REGION Network 17: ACTIVACION VAPOR VIVO Y SERPENTINA
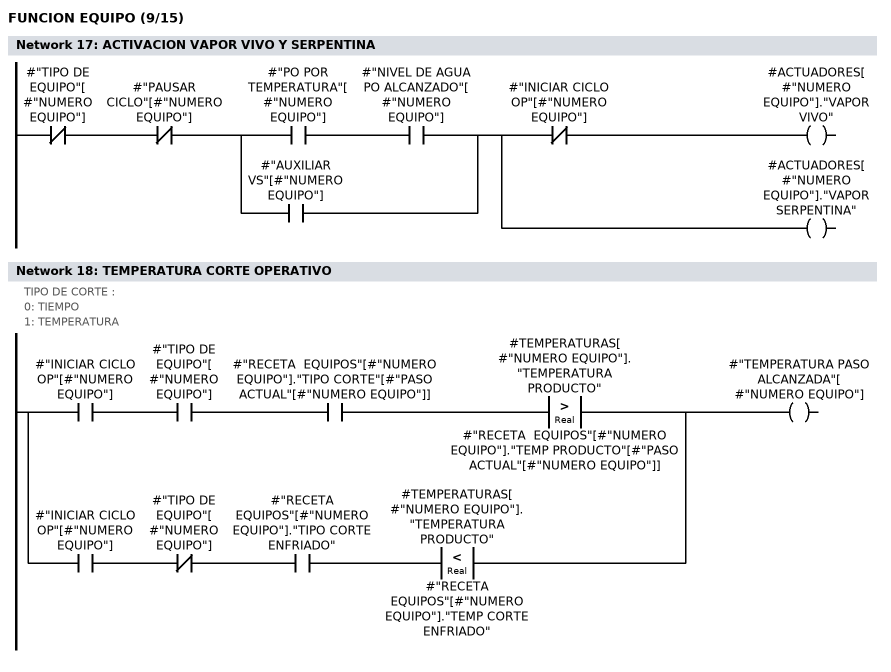
   RUNG wire#powerrail
      I_Contact( #"TIPO DE EQUIPO"[#"NUMERO EQUIPO"] )
      I_Contact( #"PAUSAR CICLO"[#"NUMERO EQUIPO"] )
      wire#w1
      Contact( #"PO POR TEMPERATURA"[#"NUMERO EQUIPO"] )
      Contact( #"NIVEL DE AGUA PO ALCANZADO"[#"NUMERO EQUIPO"] )
      wire#w2
      I_Contact( #"INICIAR CICLO OP"[#"NUMERO EQUIPO"] )
      Coil( #ACTUADORES[#"NUMERO EQUIPO"]."VAPOR VIVO" )
   END_RUNG
   RUNG wire#w1
      Contact( #"AUXILIAR VS"[#"NUMERO EQUIPO"] )
   END_RUNG wire#w2
   RUNG wire#w2
      Coil( #ACTUADORES[#"NUMERO EQUIPO"]."VAPOR SERPENTINA" )
   END_RUNG
   // the same network as SCL:
   #_w1 := NOT #"TIPO DE EQUIPO"[#"NUMERO EQUIPO"] AND NOT #"PAUSAR CICLO"[#"NUMERO EQUIPO"] AND ((#"PO POR TEMPERATURA"[#"NUMERO EQUIPO"] AND #"NIVEL DE AGUA PO ALCANZADO"[#"NUMERO EQUIPO"]) OR #"AUXILIAR VS"[#"NUMERO EQUIPO"]);
   #ACTUADORES[#"NUMERO EQUIPO"]."VAPOR VIVO" := #_w1 AND NOT #"INICIAR CICLO OP"[#"NUMERO EQUIPO"];
   #ACTUADORES[#"NUMERO EQUIPO"]."VAPOR SERPENTINA" := #_w1;
END_REGION

REGION Network 18: TEMPERATURA CORTE OPERATIVO
   // TIPO DE CORTE :
   // 
   // 0: TIEMPO
   // 1: TEMPERATURA
   RUNG wire#powerrail
      Contact( #"INICIAR CICLO OP"[#"NUMERO EQUIPO"] )
      Contact( #"TIPO DE EQUIPO"[#"NUMERO EQUIPO"] )
      Contact( #"RECETA  EQUIPOS"[#"NUMERO EQUIPO"]."TIPO CORTE"[#"PASO ACTUAL"[#"NUMERO EQUIPO"]] )
      { S7_Templates := "SrcType := Real" } GT_Contact(in1 := #TEMPERATURAS[#"NUMERO EQUIPO"]."TEMPERATURA PRODUCTO", in2 := #"RECETA  EQUIPOS"[#"NUMERO EQUIPO"]."TEMP PRODUCTO"[#"PASO ACTUAL"[#"NUMERO EQUIPO"]])
      wire#w1
      Coil( #"TEMPERATURA PASO ALCANZADA"[#"NUMERO EQUIPO"] )
   END_RUNG
   RUNG wire#powerrail
      Contact( #"INICIAR CICLO OP"[#"NUMERO EQUIPO"] )
      I_Contact( #"TIPO DE EQUIPO"[#"NUMERO EQUIPO"] )
      Contact( #"RECETA  EQUIPOS"[#"NUMERO EQUIPO"]."TIPO CORTE ENFRIADO" )
      { S7_Templates := "SrcType := Real" } LT_Contact(in1 := #TEMPERATURAS[#"NUMERO EQUIPO"]."TEMPERATURA PRODUCTO", in2 := #"RECETA  EQUIPOS"[#"NUMERO EQUIPO"]."TEMP CORTE ENFRIADO")
   END_RUNG wire#w1
   // the same network as SCL:
   #"TEMPERATURA PASO ALCANZADA"[#"NUMERO EQUIPO"] := (#"INICIAR CICLO OP"[#"NUMERO EQUIPO"] AND #"TIPO DE EQUIPO"[#"NUMERO EQUIPO"] AND #"RECETA  EQUIPOS"[#"NUMERO EQUIPO"]."TIPO CORTE"[#"PASO ACTUAL"[#"NUMERO EQUIPO"]] AND (#TEMPERATURAS[#"NUMERO EQUIPO"]."TEMPERATURA PRODUCTO" > #"RECETA  EQUIPOS"[#"NUMERO EQUIPO"]."TEMP PRODUCTO"[#"PASO ACTUAL"[#"NUMERO EQUIPO"]])) OR (#"INICIAR CICLO OP"[#"NUMERO EQUIPO"] AND NOT #"TIPO DE EQUIPO"[#"NUMERO EQUIPO"] AND #"RECETA  EQUIPOS"[#"NUMERO EQUIPO"]."TIPO CORTE ENFRIADO" AND (#TEMPERATURAS[#"NUMERO EQUIPO"]."TEMPERATURA PRODUCTO" < #"RECETA  EQUIPOS"[#"NUMERO EQUIPO"]."TEMP CORTE ENFRIADO"));
END_REGION

REGION Network 19: TIEMPO DE CORTE OPERATIVO
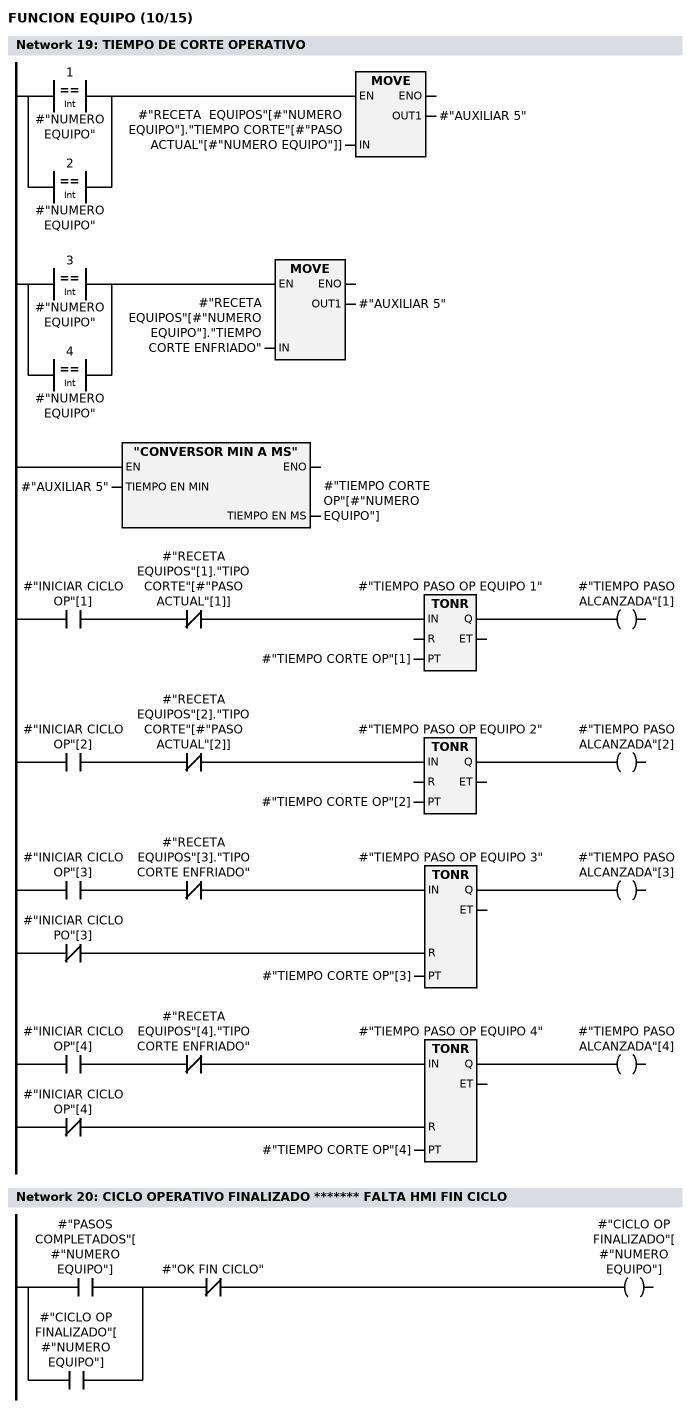
   IF (1 = #"NUMERO EQUIPO") OR (2 = #"NUMERO EQUIPO") THEN
       #"AUXILIAR 5" := #"RECETA  EQUIPOS"[#"NUMERO EQUIPO"]."TIEMPO CORTE"[#"PASO ACTUAL"[#"NUMERO EQUIPO"]];
   END_IF;
   IF (3 = #"NUMERO EQUIPO") OR (4 = #"NUMERO EQUIPO") THEN
       #"AUXILIAR 5" := #"RECETA  EQUIPOS"[#"NUMERO EQUIPO"]."TIEMPO CORTE ENFRIADO";
   END_IF;
   "CONVERSOR MIN A MS"("TIEMPO EN MIN" := #"AUXILIAR 5",
                        "TIEMPO EN MS" => #"TIEMPO CORTE OP"[#"NUMERO EQUIPO"]);
   #"TIEMPO PASO OP EQUIPO 1"(IN := #"INICIAR CICLO OP"[1] AND NOT #"RECETA  EQUIPOS"[1]."TIPO CORTE"[#"PASO ACTUAL"[1]],   // TONR
                           PT := #"TIEMPO CORTE OP"[1]);
   #"TIEMPO PASO ALCANZADA"[1] := #"TIEMPO PASO OP EQUIPO 1".Q;
   #"TIEMPO PASO OP EQUIPO 2"(IN := #"INICIAR CICLO OP"[2] AND NOT #"RECETA  EQUIPOS"[2]."TIPO CORTE"[#"PASO ACTUAL"[2]],   // TONR
                           PT := #"TIEMPO CORTE OP"[2]);
   #"TIEMPO PASO ALCANZADA"[2] := #"TIEMPO PASO OP EQUIPO 2".Q;
   #"TIEMPO PASO OP EQUIPO 3"(IN := #"INICIAR CICLO OP"[3] AND NOT #"RECETA  EQUIPOS"[3]."TIPO CORTE ENFRIADO",   // TONR
                           R := NOT #"INICIAR CICLO PO"[3],
                           PT := #"TIEMPO CORTE OP"[3]);
   #"TIEMPO PASO ALCANZADA"[3] := #"TIEMPO PASO OP EQUIPO 3".Q;
   #"TIEMPO PASO OP EQUIPO 4"(IN := #"INICIAR CICLO OP"[4] AND NOT #"RECETA  EQUIPOS"[4]."TIPO CORTE ENFRIADO",   // TONR
                           R := NOT #"INICIAR CICLO OP"[4],
                           PT := #"TIEMPO CORTE OP"[4]);
   #"TIEMPO PASO ALCANZADA"[4] := #"TIEMPO PASO OP EQUIPO 4".Q;
END_REGION

REGION Network 20: CICLO OPERATIVO FINALIZADO ******* FALTA HMI FIN CICLO
   RUNG wire#powerrail
      Contact( #"PASOS COMPLETADOS"[#"NUMERO EQUIPO"] )
      wire#w1
      I_Contact( #"OK FIN CICLO" )
      Coil( #"CICLO OP FINALIZADO"[#"NUMERO EQUIPO"] )
   END_RUNG
   RUNG wire#powerrail
      Contact( #"CICLO OP FINALIZADO"[#"NUMERO EQUIPO"] )
   END_RUNG wire#w1
   // the same network as SCL:
   #"CICLO OP FINALIZADO"[#"NUMERO EQUIPO"] := (#"PASOS COMPLETADOS"[#"NUMERO EQUIPO"] OR #"CICLO OP FINALIZADO"[#"NUMERO EQUIPO"]) AND NOT #"OK FIN CICLO";
END_REGION

REGION Network 21: CALCULO DE HISTERESIS
   // NIVEL OK
   // NIVEL BAJO
   // NIVEL ALTO
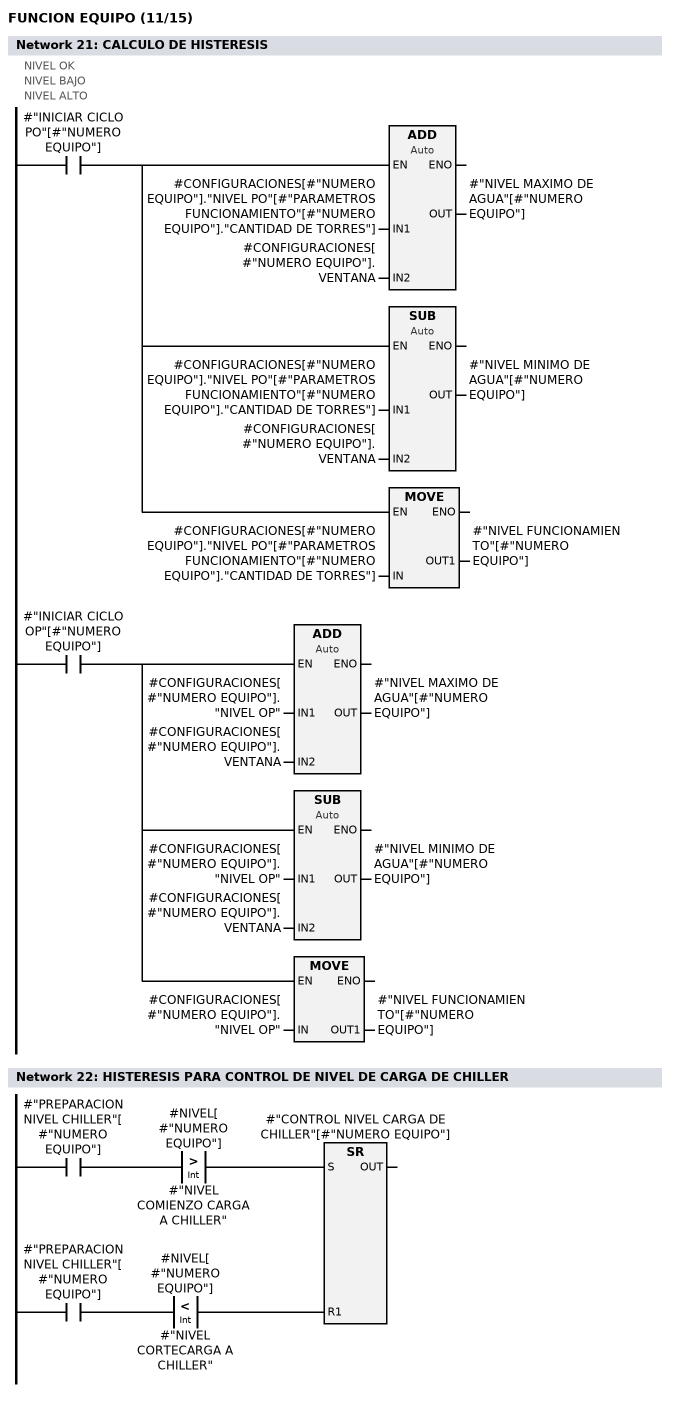
   RUNG wire#powerrail
      Contact( #"INICIAR CICLO PO"[#"NUMERO EQUIPO"] )
      wire#w1
      Add(in1 := #CONFIGURACIONES[#"NUMERO EQUIPO"]."NIVEL PO"[#"PARAMETROS FUNCIONAMIENTO"[#"NUMERO EQUIPO"]."CANTIDAD DE TORRES"], in2 := #CONFIGURACIONES[#"NUMERO EQUIPO"].VENTANA, out => #"NIVEL MAXIMO DE AGUA"[#"NUMERO EQUIPO"])
   END_RUNG
   RUNG wire#w1
      Sub(in1 := #CONFIGURACIONES[#"NUMERO EQUIPO"]."NIVEL PO"[#"PARAMETROS FUNCIONAMIENTO"[#"NUMERO EQUIPO"]."CANTIDAD DE TORRES"], in2 := #CONFIGURACIONES[#"NUMERO EQUIPO"].VENTANA, out => #"NIVEL MINIMO DE AGUA"[#"NUMERO EQUIPO"])
   END_RUNG
   RUNG wire#w1
      Move(in := #CONFIGURACIONES[#"NUMERO EQUIPO"]."NIVEL PO"[#"PARAMETROS FUNCIONAMIENTO"[#"NUMERO EQUIPO"]."CANTIDAD DE TORRES"], out1 => #"NIVEL FUNCIONAMIENTO"[#"NUMERO EQUIPO"])
   END_RUNG
   RUNG wire#powerrail
      Contact( #"INICIAR CICLO OP"[#"NUMERO EQUIPO"] )
      wire#w2
      Add(in1 := #CONFIGURACIONES[#"NUMERO EQUIPO"]."NIVEL OP", in2 := #CONFIGURACIONES[#"NUMERO EQUIPO"].VENTANA, out => #"NIVEL MAXIMO DE AGUA"[#"NUMERO EQUIPO"])
   END_RUNG
   RUNG wire#w2
      Sub(in1 := #CONFIGURACIONES[#"NUMERO EQUIPO"]."NIVEL OP", in2 := #CONFIGURACIONES[#"NUMERO EQUIPO"].VENTANA, out => #"NIVEL MINIMO DE AGUA"[#"NUMERO EQUIPO"])
   END_RUNG
   RUNG wire#w2
      Move(in := #CONFIGURACIONES[#"NUMERO EQUIPO"]."NIVEL OP", out1 => #"NIVEL FUNCIONAMIENTO"[#"NUMERO EQUIPO"])
   END_RUNG
   // the same network as SCL:
   #_w1 := #"INICIAR CICLO PO"[#"NUMERO EQUIPO"];
   IF #_w1 THEN
       #"NIVEL MAXIMO DE AGUA"[#"NUMERO EQUIPO"] := #CONFIGURACIONES[#"NUMERO EQUIPO"]."NIVEL PO"[#"PARAMETROS FUNCIONAMIENTO"[#"NUMERO EQUIPO"]."CANTIDAD DE TORRES"] + #CONFIGURACIONES[#"NUMERO EQUIPO"].VENTANA;
       #"NIVEL MINIMO DE AGUA"[#"NUMERO EQUIPO"] := #CONFIGURACIONES[#"NUMERO EQUIPO"]."NIVEL PO"[#"PARAMETROS FUNCIONAMIENTO"[#"NUMERO EQUIPO"]."CANTIDAD DE TORRES"] - #CONFIGURACIONES[#"NUMERO EQUIPO"].VENTANA;
       #"NIVEL FUNCIONAMIENTO"[#"NUMERO EQUIPO"] := #CONFIGURACIONES[#"NUMERO EQUIPO"]."NIVEL PO"[#"PARAMETROS FUNCIONAMIENTO"[#"NUMERO EQUIPO"]."CANTIDAD DE TORRES"];
   END_IF;
   #_w2 := #"INICIAR CICLO OP"[#"NUMERO EQUIPO"];
   IF #_w2 THEN
       #"NIVEL MAXIMO DE AGUA"[#"NUMERO EQUIPO"] := #CONFIGURACIONES[#"NUMERO EQUIPO"]."NIVEL OP" + #CONFIGURACIONES[#"NUMERO EQUIPO"].VENTANA;
       #"NIVEL MINIMO DE AGUA"[#"NUMERO EQUIPO"] := #CONFIGURACIONES[#"NUMERO EQUIPO"]."NIVEL OP" - #CONFIGURACIONES[#"NUMERO EQUIPO"].VENTANA;
       #"NIVEL FUNCIONAMIENTO"[#"NUMERO EQUIPO"] := #CONFIGURACIONES[#"NUMERO EQUIPO"]."NIVEL OP";
   END_IF;
END_REGION

REGION Network 22: HISTERESIS PARA CONTROL DE NIVEL DE CARGA DE CHILLER
   RUNG wire#powerrail
      Contact( #"PREPARACION NIVEL CHILLER"[#"NUMERO EQUIPO"] )
      { S7_Templates := "SrcType := Int" } GT_Contact(in1 := #NIVEL[#"NUMERO EQUIPO"], in2 := #"NIVEL COMIENZO CARGA A CHILLER")
      S_SR(operand := #"CONTROL NIVEL CARGA DE CHILLER"[#"NUMERO EQUIPO"], r1 := wire#w1)
   END_RUNG
   RUNG wire#powerrail
      Contact( #"PREPARACION NIVEL CHILLER"[#"NUMERO EQUIPO"] )
      { S7_Templates := "SrcType := Int" } LT_Contact(in1 := #NIVEL[#"NUMERO EQUIPO"], in2 := #"NIVEL CORTECARGA A CHILLER")
   END_RUNG wire#w1
   // the same network as SCL:
   #_w1 := #"PREPARACION NIVEL CHILLER"[#"NUMERO EQUIPO"] AND (#NIVEL[#"NUMERO EQUIPO"] < #"NIVEL CORTECARGA A CHILLER");
   IF #"PREPARACION NIVEL CHILLER"[#"NUMERO EQUIPO"] AND (#NIVEL[#"NUMERO EQUIPO"] > #"NIVEL COMIENZO CARGA A CHILLER") THEN
       #"CONTROL NIVEL CARGA DE CHILLER"[#"NUMERO EQUIPO"] := TRUE;   // SR flip-flop
   END_IF;
   IF #_w1 THEN #"CONTROL NIVEL CARGA DE CHILLER"[#"NUMERO EQUIPO"] := FALSE; END_IF;
END_REGION

REGION Network 23: CONTROL DE NIVEL DE AGUA DE TANQUE
   // LO CONTROLO CON UN SET Y RESET
   // 
   // 1 SR : BOMBA EGRESO
   // 2 SR : BOMBA INGRESO
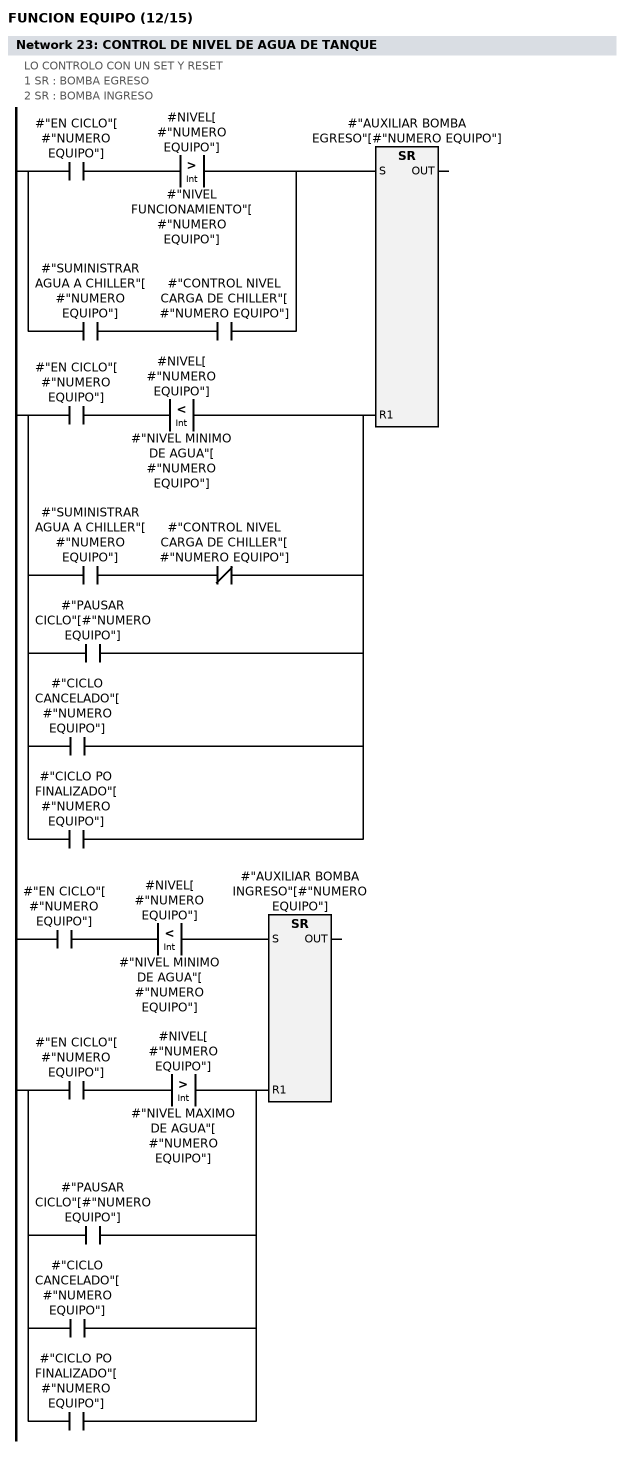
   RUNG wire#powerrail
      Contact( #"EN CICLO"[#"NUMERO EQUIPO"] )
      { S7_Templates := "SrcType := Int" } GT_Contact(in1 := #NIVEL[#"NUMERO EQUIPO"], in2 := #"NIVEL FUNCIONAMIENTO"[#"NUMERO EQUIPO"])
      wire#w1
      S_SR(operand := #"AUXILIAR BOMBA EGRESO"[#"NUMERO EQUIPO"], r1 := wire#w2)
   END_RUNG
   RUNG wire#powerrail
      Contact( #"SUMINISTRAR AGUA A CHILLER"[#"NUMERO EQUIPO"] )
      Contact( #"CONTROL NIVEL CARGA DE CHILLER"[#"NUMERO EQUIPO"] )
   END_RUNG wire#w1
   RUNG wire#powerrail
      Contact( #"EN CICLO"[#"NUMERO EQUIPO"] )
      { S7_Templates := "SrcType := Int" } LT_Contact(in1 := #NIVEL[#"NUMERO EQUIPO"], in2 := #"NIVEL MINIMO DE AGUA"[#"NUMERO EQUIPO"])
   END_RUNG wire#w2
   RUNG wire#powerrail
      Contact( #"SUMINISTRAR AGUA A CHILLER"[#"NUMERO EQUIPO"] )
      I_Contact( #"CONTROL NIVEL CARGA DE CHILLER"[#"NUMERO EQUIPO"] )
   END_RUNG wire#w2
   RUNG wire#powerrail
      Contact( #"PAUSAR CICLO"[#"NUMERO EQUIPO"] )
   END_RUNG wire#w2
   RUNG wire#powerrail
      Contact( #"CICLO CANCELADO"[#"NUMERO EQUIPO"] )
   END_RUNG wire#w2
   RUNG wire#powerrail
      Contact( #"CICLO PO FINALIZADO"[#"NUMERO EQUIPO"] )
   END_RUNG wire#w2
   RUNG wire#powerrail
      Contact( #"EN CICLO"[#"NUMERO EQUIPO"] )
      { S7_Templates := "SrcType := Int" } LT_Contact(in1 := #NIVEL[#"NUMERO EQUIPO"], in2 := #"NIVEL MINIMO DE AGUA"[#"NUMERO EQUIPO"])
      S_SR(operand := #"AUXILIAR BOMBA INGRESO"[#"NUMERO EQUIPO"], r1 := wire#w3)
   END_RUNG
   RUNG wire#powerrail
      Contact( #"EN CICLO"[#"NUMERO EQUIPO"] )
      { S7_Templates := "SrcType := Int" } GT_Contact(in1 := #NIVEL[#"NUMERO EQUIPO"], in2 := #"NIVEL MAXIMO DE AGUA"[#"NUMERO EQUIPO"])
   END_RUNG wire#w3
   RUNG wire#powerrail
      Contact( #"PAUSAR CICLO"[#"NUMERO EQUIPO"] )
   END_RUNG wire#w3
   RUNG wire#powerrail
      Contact( #"CICLO CANCELADO"[#"NUMERO EQUIPO"] )
   END_RUNG wire#w3
   RUNG wire#powerrail
      Contact( #"CICLO PO FINALIZADO"[#"NUMERO EQUIPO"] )
   END_RUNG wire#w3
   // the same network as SCL:
   #_w1 := (#"EN CICLO"[#"NUMERO EQUIPO"] AND (#NIVEL[#"NUMERO EQUIPO"] < #"NIVEL MINIMO DE AGUA"[#"NUMERO EQUIPO"])) OR (#"SUMINISTRAR AGUA A CHILLER"[#"NUMERO EQUIPO"] AND NOT #"CONTROL NIVEL CARGA DE CHILLER"[#"NUMERO EQUIPO"]) OR #"PAUSAR CICLO"[#"NUMERO EQUIPO"] OR #"CICLO CANCELADO"[#"NUMERO EQUIPO"] OR #"CICLO PO FINALIZADO"[#"NUMERO EQUIPO"];
   IF (#"EN CICLO"[#"NUMERO EQUIPO"] AND (#NIVEL[#"NUMERO EQUIPO"] > #"NIVEL FUNCIONAMIENTO"[#"NUMERO EQUIPO"])) OR (#"SUMINISTRAR AGUA A CHILLER"[#"NUMERO EQUIPO"] AND #"CONTROL NIVEL CARGA DE CHILLER"[#"NUMERO EQUIPO"]) THEN
       #"AUXILIAR BOMBA EGRESO"[#"NUMERO EQUIPO"] := TRUE;   // SR flip-flop
   END_IF;
   IF #_w1 THEN #"AUXILIAR BOMBA EGRESO"[#"NUMERO EQUIPO"] := FALSE; END_IF;
   #_w2 := (#"EN CICLO"[#"NUMERO EQUIPO"] AND (#NIVEL[#"NUMERO EQUIPO"] > #"NIVEL MAXIMO DE AGUA"[#"NUMERO EQUIPO"])) OR #"PAUSAR CICLO"[#"NUMERO EQUIPO"] OR #"CICLO CANCELADO"[#"NUMERO EQUIPO"] OR #"CICLO PO FINALIZADO"[#"NUMERO EQUIPO"];
   IF #"EN CICLO"[#"NUMERO EQUIPO"] AND (#NIVEL[#"NUMERO EQUIPO"] < #"NIVEL MINIMO DE AGUA"[#"NUMERO EQUIPO"]) THEN
       #"AUXILIAR BOMBA INGRESO"[#"NUMERO EQUIPO"] := TRUE;   // SR flip-flop
   END_IF;
   IF #_w2 THEN #"AUXILIAR BOMBA INGRESO"[#"NUMERO EQUIPO"] := FALSE; END_IF;
END_REGION

REGION Network 24: DELAY ENTRE VALVULAS Y BOMBAS DE INGRESO Y EGRESO
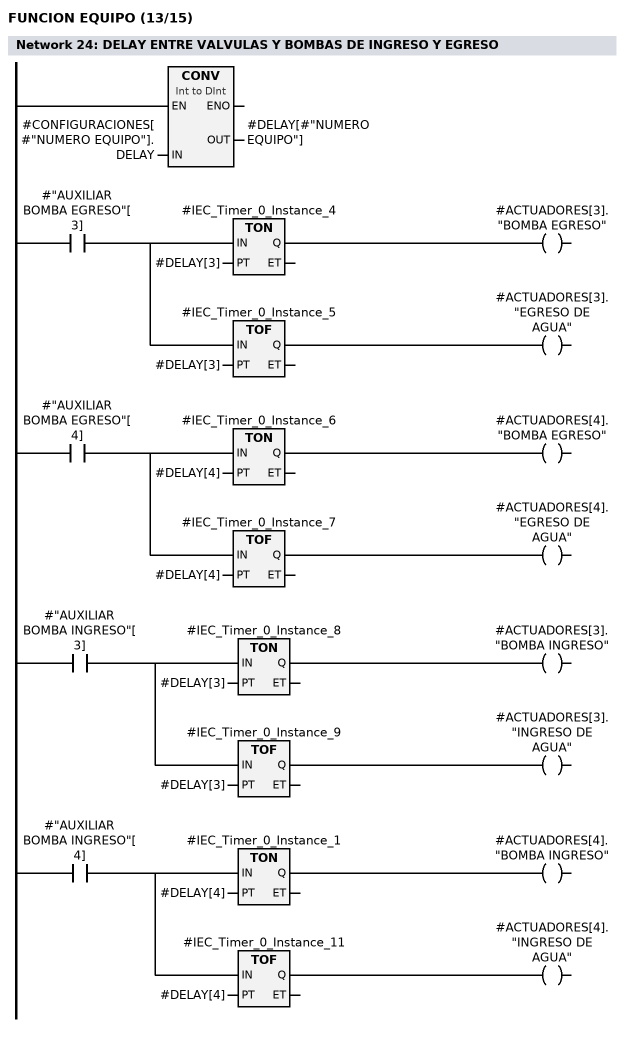
   #DELAY[#"NUMERO EQUIPO"] := INT_TO_DINT(#CONFIGURACIONES[#"NUMERO EQUIPO"].DELAY);
   #IEC_Timer_0_Instance_4(IN := #"AUXILIAR BOMBA EGRESO"[3], PT := #DELAY[3]);   // TON
   #ACTUADORES[3]."BOMBA EGRESO" := #IEC_Timer_0_Instance_4.Q;
   #IEC_Timer_0_Instance_5(IN := #"AUXILIAR BOMBA EGRESO"[3], PT := #DELAY[3]);   // TOF
   #ACTUADORES[3]."EGRESO DE AGUA" := #IEC_Timer_0_Instance_5.Q;
   #IEC_Timer_0_Instance_6(IN := #"AUXILIAR BOMBA EGRESO"[4], PT := #DELAY[4]);   // TON
   #ACTUADORES[4]."BOMBA EGRESO" := #IEC_Timer_0_Instance_6.Q;
   #IEC_Timer_0_Instance_7(IN := #"AUXILIAR BOMBA EGRESO"[4], PT := #DELAY[4]);   // TOF
   #ACTUADORES[4]."EGRESO DE AGUA" := #IEC_Timer_0_Instance_7.Q;
   #IEC_Timer_0_Instance_8(IN := #"AUXILIAR BOMBA INGRESO"[3], PT := #DELAY[3]);   // TON
   #ACTUADORES[3]."BOMBA INGRESO" := #IEC_Timer_0_Instance_8.Q;
   #IEC_Timer_0_Instance_9(IN := #"AUXILIAR BOMBA INGRESO"[3], PT := #DELAY[3]);   // TOF
   #ACTUADORES[3]."INGRESO DE AGUA" := #IEC_Timer_0_Instance_9.Q;
   #IEC_Timer_0_Instance_1(IN := #"AUXILIAR BOMBA INGRESO"[4], PT := #DELAY[4]);   // TON
   #ACTUADORES[4]."BOMBA INGRESO" := #IEC_Timer_0_Instance_1.Q;
   #IEC_Timer_0_Instance_11(IN := #"AUXILIAR BOMBA INGRESO"[4], PT := #DELAY[4]);   // TOF
   #ACTUADORES[4]."INGRESO DE AGUA" := #IEC_Timer_0_Instance_11.Q;
END_REGION

REGION Network 25: NIVELES DE CHILLER
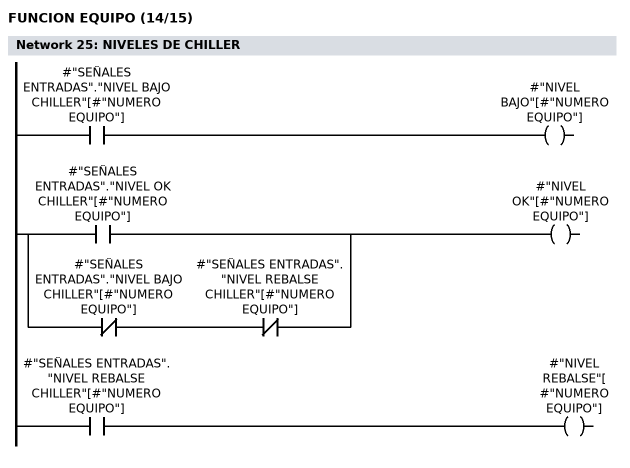
   RUNG wire#powerrail
      Contact( #"SEÑALES ENTRADAS"."NIVEL BAJO CHILLER"[#"NUMERO EQUIPO"] )
      Coil( #"NIVEL BAJO"[#"NUMERO EQUIPO"] )
   END_RUNG
   RUNG wire#powerrail
      Contact( #"SEÑALES ENTRADAS"."NIVEL OK CHILLER"[#"NUMERO EQUIPO"] )
      wire#w1
      Coil( #"NIVEL OK"[#"NUMERO EQUIPO"] )
   END_RUNG
   RUNG wire#powerrail
      I_Contact( #"SEÑALES ENTRADAS"."NIVEL BAJO CHILLER"[#"NUMERO EQUIPO"] )
      I_Contact( #"SEÑALES ENTRADAS"."NIVEL REBALSE CHILLER"[#"NUMERO EQUIPO"] )
   END_RUNG wire#w1
   RUNG wire#powerrail
      Contact( #"SEÑALES ENTRADAS"."NIVEL REBALSE CHILLER"[#"NUMERO EQUIPO"] )
      Coil( #"NIVEL REBALSE"[#"NUMERO EQUIPO"] )
   END_RUNG
   // the same network as SCL:
   #"NIVEL BAJO"[#"NUMERO EQUIPO"] := #"SEÑALES ENTRADAS"."NIVEL BAJO CHILLER"[#"NUMERO EQUIPO"];
   #"NIVEL OK"[#"NUMERO EQUIPO"] := #"SEÑALES ENTRADAS"."NIVEL OK CHILLER"[#"NUMERO EQUIPO"] OR (NOT #"SEÑALES ENTRADAS"."NIVEL BAJO CHILLER"[#"NUMERO EQUIPO"] AND NOT #"SEÑALES ENTRADAS"."NIVEL REBALSE CHILLER"[#"NUMERO EQUIPO"]);
   #"NIVEL REBALSE"[#"NUMERO EQUIPO"] := #"SEÑALES ENTRADAS"."NIVEL REBALSE CHILLER"[#"NUMERO EQUIPO"];
END_REGION

REGION Network 26: PASE DE ESTADOS
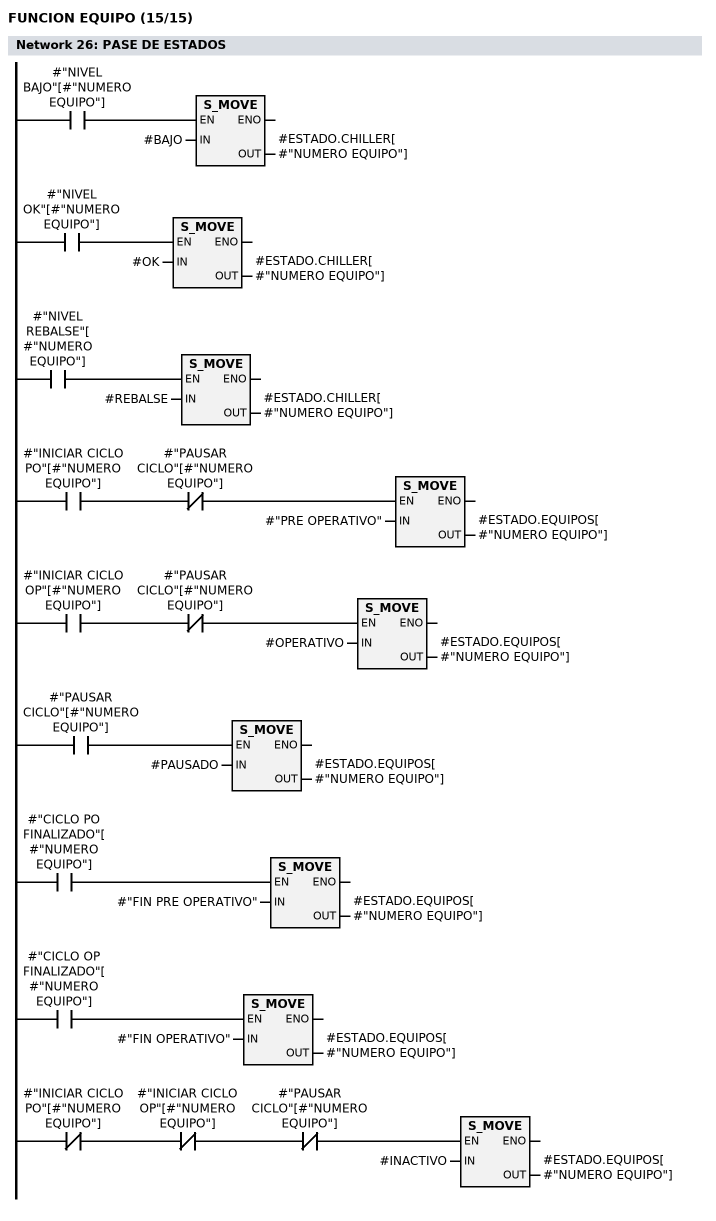
   RUNG wire#powerrail
      Contact( #"NIVEL BAJO"[#"NUMERO EQUIPO"] )
      S_Move(in := #BAJO, out => #ESTADO.CHILLER[#"NUMERO EQUIPO"])
   END_RUNG
   RUNG wire#powerrail
      Contact( #"NIVEL OK"[#"NUMERO EQUIPO"] )
      S_Move(in := #OK, out => #ESTADO.CHILLER[#"NUMERO EQUIPO"])
   END_RUNG
   RUNG wire#powerrail
      Contact( #"NIVEL REBALSE"[#"NUMERO EQUIPO"] )
      S_Move(in := #REBALSE, out => #ESTADO.CHILLER[#"NUMERO EQUIPO"])
   END_RUNG
   RUNG wire#powerrail
      Contact( #"INICIAR CICLO PO"[#"NUMERO EQUIPO"] )
      I_Contact( #"PAUSAR CICLO"[#"NUMERO EQUIPO"] )
      S_Move(in := #"PRE OPERATIVO", out => #ESTADO.EQUIPOS[#"NUMERO EQUIPO"])
   END_RUNG
   RUNG wire#powerrail
      Contact( #"INICIAR CICLO OP"[#"NUMERO EQUIPO"] )
      I_Contact( #"PAUSAR CICLO"[#"NUMERO EQUIPO"] )
      S_Move(in := #OPERATIVO, out => #ESTADO.EQUIPOS[#"NUMERO EQUIPO"])
   END_RUNG
   RUNG wire#powerrail
      Contact( #"PAUSAR CICLO"[#"NUMERO EQUIPO"] )
      S_Move(in := #PAUSADO, out => #ESTADO.EQUIPOS[#"NUMERO EQUIPO"])
   END_RUNG
   RUNG wire#powerrail
      Contact( #"CICLO PO FINALIZADO"[#"NUMERO EQUIPO"] )
      S_Move(in := #"FIN PRE OPERATIVO", out => #ESTADO.EQUIPOS[#"NUMERO EQUIPO"])
   END_RUNG
   RUNG wire#powerrail
      Contact( #"CICLO OP FINALIZADO"[#"NUMERO EQUIPO"] )
      S_Move(in := #"FIN OPERATIVO", out => #ESTADO.EQUIPOS[#"NUMERO EQUIPO"])
   END_RUNG
   RUNG wire#powerrail
      I_Contact( #"INICIAR CICLO PO"[#"NUMERO EQUIPO"] )
      I_Contact( #"INICIAR CICLO OP"[#"NUMERO EQUIPO"] )
      I_Contact( #"PAUSAR CICLO"[#"NUMERO EQUIPO"] )
      S_Move(in := #INACTIVO, out => #ESTADO.EQUIPOS[#"NUMERO EQUIPO"])
   END_RUNG
   // the same network as SCL:
   IF #"NIVEL BAJO"[#"NUMERO EQUIPO"] THEN #ESTADO.CHILLER[#"NUMERO EQUIPO"] := #BAJO; END_IF;
   IF #"NIVEL OK"[#"NUMERO EQUIPO"] THEN #ESTADO.CHILLER[#"NUMERO EQUIPO"] := #OK; END_IF;
   IF #"NIVEL REBALSE"[#"NUMERO EQUIPO"] THEN #ESTADO.CHILLER[#"NUMERO EQUIPO"] := #REBALSE; END_IF;
   IF #"INICIAR CICLO PO"[#"NUMERO EQUIPO"] AND NOT #"PAUSAR CICLO"[#"NUMERO EQUIPO"] THEN
       #ESTADO.EQUIPOS[#"NUMERO EQUIPO"] := #"PRE OPERATIVO";
   END_IF;
   IF #"INICIAR CICLO OP"[#"NUMERO EQUIPO"] AND NOT #"PAUSAR CICLO"[#"NUMERO EQUIPO"] THEN
       #ESTADO.EQUIPOS[#"NUMERO EQUIPO"] := #OPERATIVO;
   END_IF;
   IF #"PAUSAR CICLO"[#"NUMERO EQUIPO"] THEN #ESTADO.EQUIPOS[#"NUMERO EQUIPO"] := #PAUSADO; END_IF;
   IF #"CICLO PO FINALIZADO"[#"NUMERO EQUIPO"] THEN
       #ESTADO.EQUIPOS[#"NUMERO EQUIPO"] := #"FIN PRE OPERATIVO";
   END_IF;
   IF #"CICLO OP FINALIZADO"[#"NUMERO EQUIPO"] THEN
       #ESTADO.EQUIPOS[#"NUMERO EQUIPO"] := #"FIN OPERATIVO";
   END_IF;
   IF NOT #"INICIAR CICLO PO"[#"NUMERO EQUIPO"] AND NOT #"INICIAR CICLO OP"[#"NUMERO EQUIPO"] AND NOT #"PAUSAR CICLO"[#"NUMERO EQUIPO"] THEN
       #ESTADO.EQUIPOS[#"NUMERO EQUIPO"] := #INACTIVO;
   END_IF;
END_REGION
END_FUNCTION_BLOCK

FUNCTION_BLOCK "COCINA"   // FB5, LAD
{ S7_Optimized_Access := 'TRUE' }
VERSION : 0.1
   VAR_INPUT
      REARME : Bool;
      "PARAMETROS CICLOS" : Struct
         "CANTIDAD DE TORRES" : Int;
         "NIVEL MINIMO" : Array[1..3] of Int;   // El arreglo es porque hay 3 torres
         "TIPO DE CORTE" : Bool;
         "TEMPERATURA CORTE PO" : Int;
         "TIEMPO CORTE PO" : Int;
         "NUMERO RECETA" : Int;
         "NOMBRE RECETA" : String;
         "ESTADO ACTUAL" : String;
         "TIEMPO TOTAL TRANSCURRIDO" : Int;
         "PASO ACTUAL" : Int;
         "VAPOR VIVO" : Bool;
      END_STRUCT;
      CONFIGURACION : Struct
         DELAY : Int;
         HISTERESIS : DInt;
         "TIEMPO MAXIMO CICLO" : Int;
         "NIVEL CRITICO" : Int;
         "NIVEL PO" : Array[1..3] of Int;
         "NIVEL OP" : Int;
         VENTANA : Int;
         "NIVEL CRITICO OP" : Int;
      END_STRUCT;
      RECETA : Struct
         PASOS : Int;
         "TEMP AGUA" : Array[1..4] of Int;
         "TEMP PRODUCTO" : Array[1..4] of Int;
         "TIEMPO CORTE" : Array[1..4] of Int;
         "TIPO CORTE" : Array[1..4] of Bool;
         NOMBRE : String;
         "TIEMPO CORTE ENFRIADO" : Int;
         "TEMP CORTE ENFRIADO" : Int;
         "TIPO CORTE ENFRIADO" : Bool;
      END_STRUCT;
      TEMPERATURAS : Struct
         "TEMPERATURA AGUA" : Real;
         "TEMPERATURA INGRESO" : Real;
         "TEMPERATURA PRODUCTO" : Real;
         "TEMPERATURA AGUA SC" : Real;
         "TEMPERATURA INGRESO SC" : Real;
         "TEMPERATURA PRODUCTO SC" : Real;
      END_STRUCT;
      NIVEL : Int;
      GUARDAMOTOR : Bool;
      "VAPOR VIVO CERRADO" : Bool;
      "VAPOR VIVO ABIERTO" : Bool;
      "SERPENTINA CERRADA" : Bool;
      "SERPENTINA ABIERTA" : Bool;
      "MANUAL VAPOR VIVO" : Bool;
      "MANUAL VAPOR SERPENTINA" : Bool;
      "MANUAL CARGA DE AGUA" : Bool;
      "MANUAL TOMA FILTRO" : Bool;
      "MANUAL BOMBA" : Bool;
      "MANUAL BALIZA VERDE" : Bool;
      "MANUAL BALIZA ROJA" : Bool;
      "MANUAL LEVANTAR TAPA" : Bool;
      "MANUAL BAJAR TAPA" : Bool;
      "EQUIPO SELECCIONADO" : Int;
      "NUMERO DE EQUIPO" : Int;
      "SALTAR PASO" : Bool;
      "INICIAR PRE OPERATIVO" : Bool;
      "INICIAR OPERATIVO" : Bool;
      PAUSA : Bool;
      CONTINUAR : Bool;
      CANCELAR : Bool;
      "PULSADOR EMERGENCIA" : Bool;
      "OK FIN CICLO" : Bool;
      "OK CANCELAR" : Bool;
      "RESET ACTUADORES MANUAL" : Bool;
      "CONFIRMAR LOTE" : Bool;
   END_VAR
   VAR_OUTPUT
      "BALIZA VERDE" : Bool;
      "BALIZA ROJA" : Bool;
      BUZER : Bool;
      BOMBA : Bool;
      "CARGA DE AGUA" : Bool;
      "TOMA FILTRO" : Bool;
      "VAPOR SERPENTINA" : Bool;
      "VAPOR VIVO" : Bool;
      ESTADO : Struct
         EQUIPO : String;
         CHILLER : String;
         "COLOR EN HMI" : Int;
         "TIEMPO TRANSCURRIDO" : DInt;
         "EN PO" : Bool;
         "EN OP" : Bool;
         "EN CICLO" : Bool;
         "TIPO DE CORTE" : String;
         "PULSADOR PAUSA" : Bool;
         "PULSADOR CONTINUAR" : Bool;
         "PULSADOR CANCELAR" : Bool;
         "CICLO CANCELADO" : Bool;
         "CICLO FINALIZADO" : Bool;
         "PULSADOR CICLO CANCELADO" : Bool;
         "PULSADOR CICLO FINALIZADO" : Bool;
         "RESET ACTUADORES" : Bool;
         "MANUAL ACTIVO" : Bool;
         "PASO ACTUAL" : Int;
         "CONFIRMACION LOTE" : Bool;
      END_STRUCT;
      ALARMAS : Struct
         "FALLA VALVULA VAPOR SERPENTINA" : Bool;
         "FALLA VALVULA VAPOR VIVO" : Bool;
         "FALLA GUARDAMOTOR" : Bool;
         "NIVEL CRITICO" : Bool;
         "FALLA SENSOR TEMP AGUA" : Bool;
         "FALLA SENSOR TEMP INGRESO" : Bool;
         "FALLA SENSOR TEMP PRODUCTO" : Bool;
         "TIEMPO MAXIMO CARGA DE AGUA" : Bool;
      END_STRUCT;
      "ESTADO SALIDAS" : Struct
         "BALIZA VERDE" : Bool;
         "BALIZA ROJA" : Bool;
         BOMBA : Bool;
         "CARGA DE GUA" : Bool;
         "TOMA FILTRO" : Bool;
         "VAPOR SERPENTINA" : Bool;
         "VAPOR VIVO" : Bool;
      END_STRUCT;
      "ESTADO ENTRADAS" : Struct
         GUARDAMOTOR : Bool;
         "VAPOR VIVO CERRADO" : Bool;
         "VAPOR VIVO ABIERTO" : Bool;
         "SERPENTINA CERRADA" : Bool;
         "SERPENTINA ABIERTA" : Bool;
      END_STRUCT;
   END_VAR
   VAR
      HABILITADO : Bool;
      "EN FALLA" : Bool;
      "CICLO CANCELADO" : Bool;
      "CICLO PAUSADO" : Bool;
      "CICLO PO ACTIVO" : Bool;
      "CICLO OP ACTIVO" : Bool;
      "FIN CICLO PO" : Bool;
      "NIVEL PO" : Int;
      "NIVEL TQ ALCANZADO" : Bool;
      "CARGA AGUA TQ" : Bool;
      "NIVEL PARA CARGA DE AGUA" : Int;
      "TEMPERATURA PO ALCANZADA" : Bool;
      "TIEMPO PO ALCANZADO" : Bool;
      "TIEMPO CORTE PO" : DInt;
      IEC_Timer_0_Instance : TONR_TIME;
      "FIN CICLO OP" : Bool;
      IEC_Counter_0_Instance : CTU_INT;
      "PASO ACTUAL" : Int;
      AUXILIAR : Int;
      "TEMPERATURA PASO ALCANZADA" : Bool;
      IEC_Timer_0_Instance_1 : TONR_TIME;
      "TIEMPO PASO ALCANZADO" : Bool;
      "TIEMPO DE PASO EN OP" : DInt;
      "TEMP MAXIMA" : Real;
      "TEMP MINIMA" : Real;
      "TEMP EN RANGO" : Bool;
      "TEMP BAJA" : Bool;
      "TEMP ALTA" : Bool;
      "CICLO PO FINALIZADO" : Bool;
      "CICLO OP FINALIZADO" : Bool;
      IEC_Timer_0_Instance_2 : TON_TIME;
      IEC_Timer_0_Instance_3 : TON_TIME;
      "FALLA VALVULA SERPENTINA" : Bool;
      "FALLA CIERRE VS" : Bool;
      "FALLA VALVULA VAPOR VIVO" : Bool;
      "FALLA CIERRE VV" : Bool;
      IEC_Timer_0_Instance_4 : TON_TIME;
      IEC_Timer_0_Instance_5 : TON_TIME;
      "SE ALCANZO UN NIVEL CRITICO" : Bool;
      F1 : Bool;
      "FALLA SENSOR TEMPERATURA" : Bool;
      IEC_Timer_0_Instance_6 : TONR_TIME;
      IEC_Timer_0_Instance_7 : TON_TIME;
      IEC_Timer_0_Instance_8 : TON_TIME;
      IEC_Timer_0_Instance_9 : TONR_TIME;
      "TIEMPO MAXIMO" : DInt;
      "AUXILIAR TIEMPO" : DInt;
      IEC_Timer_0_Instance_10 : TONR_TIME;
      "TIEMPO MAXIMO CARGA DE AGUA" : Bool;
      "NIVEL CRITICO PO" : Bool;
      "NIVEL CRITICO OP" : Bool;
      "CONTINUAR CICLO" : Bool;
      IEC_Timer_0_Instance_11 : TOF_TIME;
      F5 : Bool;
      F6 : Bool;
      F7 : Bool;
      F8 : Bool;
      "TEMP MAXIMA CHILLER" : Real;
      "TEMP MINIMA CHILLER" : Real;
      "TEMP ALTA CHILLER" : Bool;
      "TEMP BAJA CHILLER" : Bool;
      "TEMP EN RANGO CHILLER" : Bool;
      IEC_Timer_0_Instance_12 : TOF_TIME;
      F9 : Bool;
      "PREPARACION FRIO CHILLER EN COCCION" : Bool;
      "PREPARACION FRIO CHILLER EN ENFRIADO" : Bool;
      "SALIDA AUX 1 CLIENTE" : Bool;
      "SALIDA AUX 2 CLIENTE" : Bool;
      "CONFIRMAR LOTE_1" : Bool;
   END_VAR
   VAR CONSTANT
      "MAXIMO APERTURA VALVULAS" : Time := T#7S;
      TEMPERATURA : String := 'TEMPERATURA';
      TIEMPO : String := 'TIEMPO';
      "PRE OPERACIONAL" : String := 'PRE OPERACIONAL';
      OPERACIONAL : String := 'OPERACIONAL';
      PAUSADO : String := 'PAUSADO';
      INACTIVO : String := 'INACTIVO';
      CANCELADO : String := 'CANCELADO';
      FINALIZADO : String := 'FINALIZADO';
      "NIVEL FILTRO" : Int := 980;
      "NIVEL TOMA FILTRO" : Int := 550;
   END_VAR
   VAR_TEMP   // added for the SCL form of the ladder/FBD networks
      _w1 : Bool;
      _w2 : Bool;
      _w3 : Bool;
      _w4 : Bool;
      _w5 : Bool;
   END_VAR
   // // CONFIGURACION."NIVEL PO"[1] : Nivel PO para 1 torre
   // // CONFIGURACION."NIVEL PO"[2] : Nivel PO para 2 torres
   // // CONFIGURACION."NIVEL PO"[3] : Nivel PO para 3 torres
BEGIN

REGION Network 1: HABILITACION
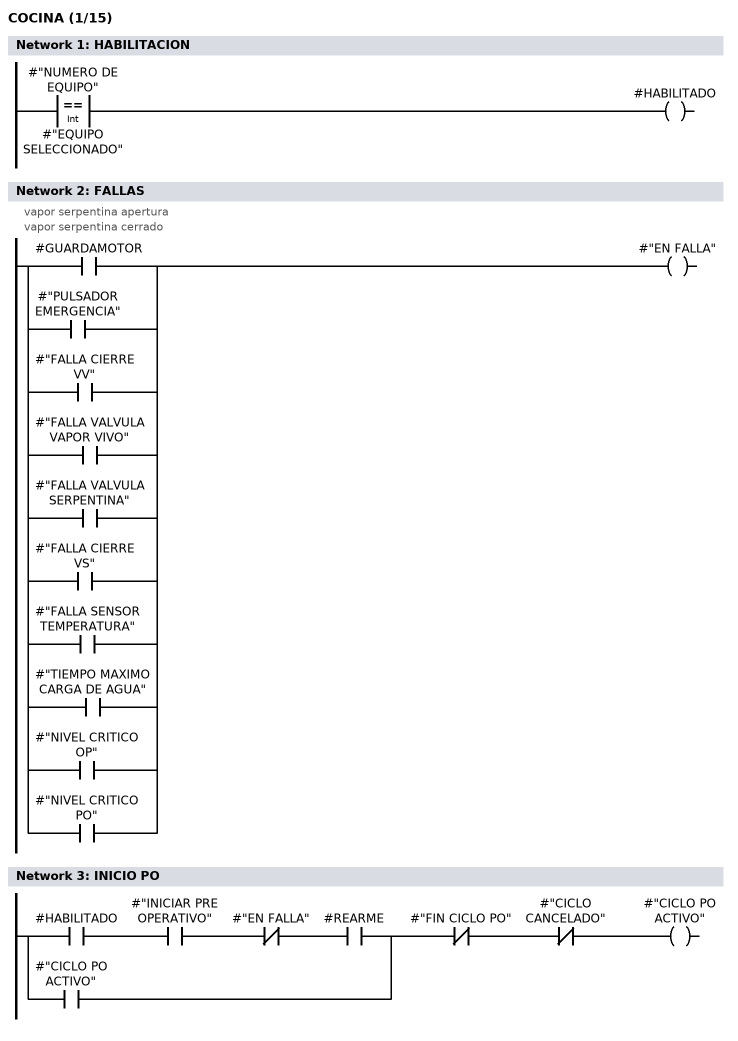
   RUNG wire#powerrail
      { S7_Templates := "SrcType := Int" } EQ_Contact(in1 := #"NUMERO DE EQUIPO", in2 := #"EQUIPO SELECCIONADO")
      Coil( #HABILITADO )
   END_RUNG
   // the same network as SCL:
   #HABILITADO := #"NUMERO DE EQUIPO" = #"EQUIPO SELECCIONADO";
END_REGION

REGION Network 2: FALLAS
   // vapor serpentina apertura
   // vapor serpentina cerrado
   RUNG wire#powerrail
      Contact( #GUARDAMOTOR )
      wire#w1
      Coil( #"EN FALLA" )
   END_RUNG
   RUNG wire#powerrail
      Contact( #"PULSADOR EMERGENCIA" )
   END_RUNG wire#w1
   RUNG wire#powerrail
      Contact( #"FALLA CIERRE VV" )
   END_RUNG wire#w1
   RUNG wire#powerrail
      Contact( #"FALLA VALVULA VAPOR VIVO" )
   END_RUNG wire#w1
   RUNG wire#powerrail
      Contact( #"FALLA VALVULA SERPENTINA" )
   END_RUNG wire#w1
   RUNG wire#powerrail
      Contact( #"FALLA CIERRE VS" )
   END_RUNG wire#w1
   RUNG wire#powerrail
      Contact( #"FALLA SENSOR TEMPERATURA" )
   END_RUNG wire#w1
   RUNG wire#powerrail
      Contact( #"TIEMPO MAXIMO CARGA DE AGUA" )
   END_RUNG wire#w1
   RUNG wire#powerrail
      Contact( #"NIVEL CRITICO OP" )
   END_RUNG wire#w1
   RUNG wire#powerrail
      Contact( #"NIVEL CRITICO PO" )
   END_RUNG wire#w1
   // the same network as SCL:
   #"EN FALLA" := #GUARDAMOTOR OR #"PULSADOR EMERGENCIA" OR #"FALLA CIERRE VV" OR #"FALLA VALVULA VAPOR VIVO" OR #"FALLA VALVULA SERPENTINA" OR #"FALLA CIERRE VS" OR #"FALLA SENSOR TEMPERATURA" OR #"TIEMPO MAXIMO CARGA DE AGUA" OR #"NIVEL CRITICO OP" OR #"NIVEL CRITICO PO";
END_REGION

REGION Network 3: INICIO PO
   RUNG wire#powerrail
      Contact( #HABILITADO )
      Contact( #"INICIAR PRE OPERATIVO" )
      I_Contact( #"EN FALLA" )
      Contact( #REARME )
      wire#w1
      I_Contact( #"FIN CICLO PO" )
      I_Contact( #"CICLO CANCELADO" )
      Coil( #"CICLO PO ACTIVO" )
   END_RUNG
   RUNG wire#powerrail
      Contact( #"CICLO PO ACTIVO" )
   END_RUNG wire#w1
   // the same network as SCL:
   #"CICLO PO ACTIVO" := ((#HABILITADO AND #"INICIAR PRE OPERATIVO" AND NOT #"EN FALLA" AND #REARME) OR #"CICLO PO ACTIVO") AND NOT #"FIN CICLO PO" AND NOT #"CICLO CANCELADO";
END_REGION

REGION Network 4: ACTIVACION CANCELACION PAUSA
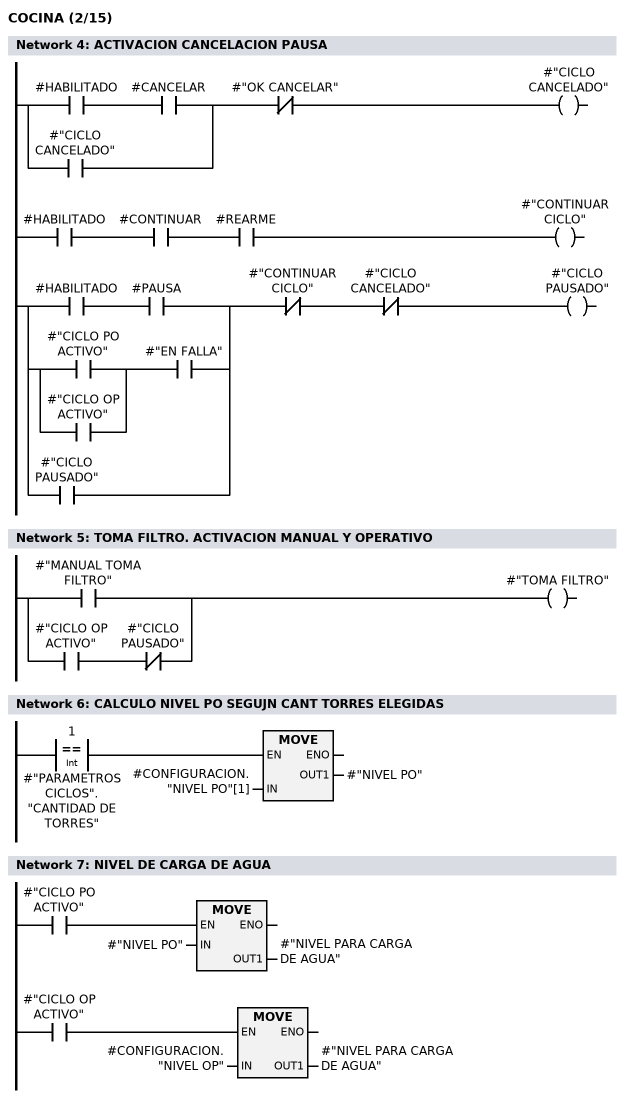
   RUNG wire#powerrail
      Contact( #HABILITADO )
      Contact( #CANCELAR )
      wire#w1
      I_Contact( #"OK CANCELAR" )
      Coil( #"CICLO CANCELADO" )
   END_RUNG
   RUNG wire#powerrail
      Contact( #"CICLO CANCELADO" )
   END_RUNG wire#w1
   RUNG wire#powerrail
      Contact( #HABILITADO )
      Contact( #CONTINUAR )
      Contact( #REARME )
      Coil( #"CONTINUAR CICLO" )
   END_RUNG
   RUNG wire#powerrail
      Contact( #HABILITADO )
      Contact( #PAUSA )
      wire#w2
      I_Contact( #"CONTINUAR CICLO" )
      I_Contact( #"CICLO CANCELADO" )
      Coil( #"CICLO PAUSADO" )
   END_RUNG
   RUNG wire#powerrail
      Contact( #"CICLO PO ACTIVO" )
      wire#w3
      Contact( #"EN FALLA" )
   END_RUNG wire#w2
   RUNG wire#powerrail
      Contact( #"CICLO OP ACTIVO" )
   END_RUNG wire#w3
   RUNG wire#powerrail
      Contact( #"CICLO PAUSADO" )
   END_RUNG wire#w2
   // the same network as SCL:
   #"CICLO CANCELADO" := ((#HABILITADO AND #CANCELAR) OR #"CICLO CANCELADO") AND NOT #"OK CANCELAR";
   #"CONTINUAR CICLO" := #HABILITADO AND #CONTINUAR AND #REARME;
   #"CICLO PAUSADO" := ((#HABILITADO AND #PAUSA) OR ((#"CICLO PO ACTIVO" OR #"CICLO OP ACTIVO") AND #"EN FALLA") OR #"CICLO PAUSADO") AND NOT #"CONTINUAR CICLO" AND NOT #"CICLO CANCELADO";
END_REGION

REGION Network 5: TOMA FILTRO. ACTIVACION MANUAL Y OPERATIVO
   RUNG wire#powerrail
      Contact( #"MANUAL TOMA FILTRO" )
      wire#w1
      Coil( #"TOMA FILTRO" )
   END_RUNG
   RUNG wire#powerrail
      Contact( #"CICLO OP ACTIVO" )
      I_Contact( #"CICLO PAUSADO" )
   END_RUNG wire#w1
   // the same network as SCL:
   #"TOMA FILTRO" := #"MANUAL TOMA FILTRO" OR (#"CICLO OP ACTIVO" AND NOT #"CICLO PAUSADO");
END_REGION

REGION Network 6: CALCULO NIVEL PO SEGUJN CANT TORRES ELEGIDAS
   RUNG wire#powerrail
      { S7_Templates := "SrcType := Int" } EQ_Contact(in1 := 1, in2 := #"PARAMETROS CICLOS"."CANTIDAD DE TORRES")
      Move(in := #CONFIGURACION."NIVEL PO"[1], out1 => #"NIVEL PO")
   END_RUNG
   // the same network as SCL:
   IF 1 = #"PARAMETROS CICLOS"."CANTIDAD DE TORRES" THEN #"NIVEL PO" := #CONFIGURACION."NIVEL PO"[1]; END_IF;
END_REGION

REGION Network 7: NIVEL DE CARGA DE AGUA
   RUNG wire#powerrail
      Contact( #"CICLO PO ACTIVO" )
      Move(in := #"NIVEL PO", out1 => #"NIVEL PARA CARGA DE AGUA")
   END_RUNG
   RUNG wire#powerrail
      Contact( #"CICLO OP ACTIVO" )
      Move(in := #CONFIGURACION."NIVEL OP", out1 => #"NIVEL PARA CARGA DE AGUA")
   END_RUNG
   // the same network as SCL:
   IF #"CICLO PO ACTIVO" THEN #"NIVEL PARA CARGA DE AGUA" := #"NIVEL PO"; END_IF;
   IF #"CICLO OP ACTIVO" THEN #"NIVEL PARA CARGA DE AGUA" := #CONFIGURACION."NIVEL OP"; END_IF;
END_REGION

REGION Network 8: BUSQUEDA DE NIVEL EN CARGA DE AGUA DE NIVEL DE TANQUE
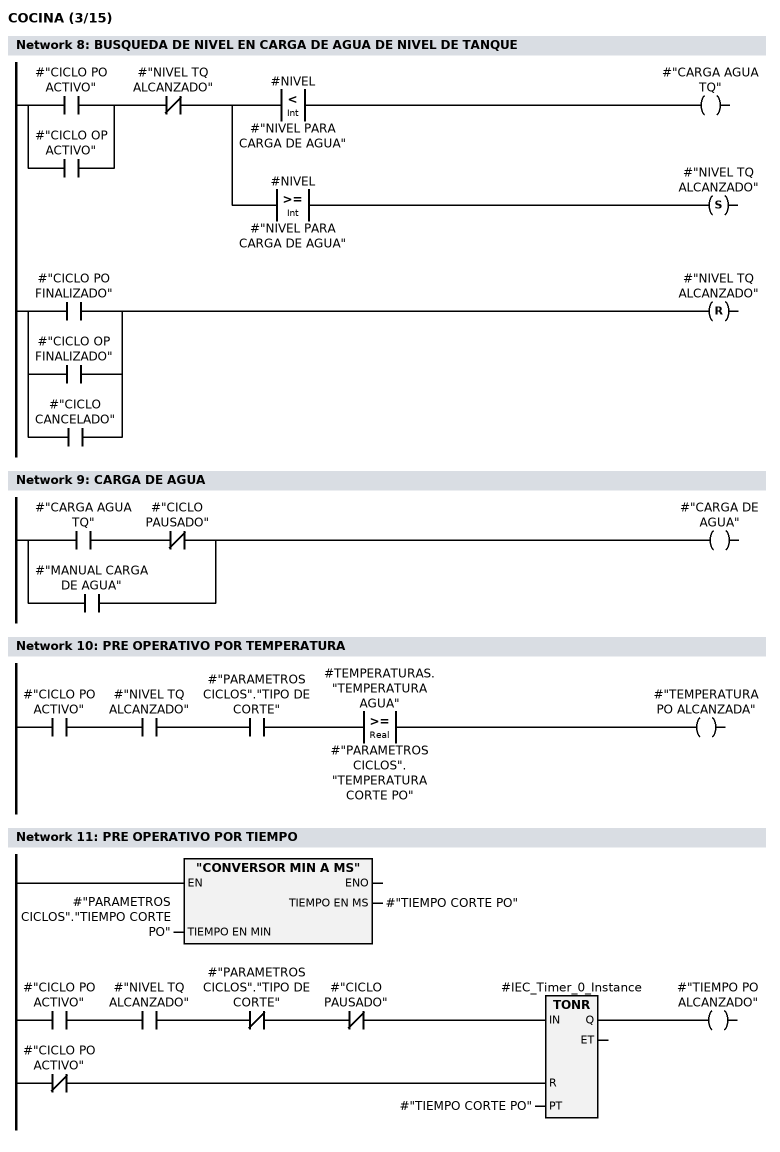
   RUNG wire#powerrail
      Contact( #"CICLO PO ACTIVO" )
      wire#w1
      I_Contact( #"NIVEL TQ ALCANZADO" )
      wire#w2
      { S7_Templates := "SrcType := Int" } LT_Contact(in1 := #NIVEL, in2 := #"NIVEL PARA CARGA DE AGUA")
      Coil( #"CARGA AGUA TQ" )
   END_RUNG
   RUNG wire#powerrail
      Contact( #"CICLO OP ACTIVO" )
   END_RUNG wire#w1
   RUNG wire#w2
      { S7_Templates := "SrcType := Int" } GE_Contact(in1 := #NIVEL, in2 := #"NIVEL PARA CARGA DE AGUA")
      S_Coil( #"NIVEL TQ ALCANZADO" )
   END_RUNG
   RUNG wire#powerrail
      Contact( #"CICLO PO FINALIZADO" )
      wire#w3
      R_Coil( #"NIVEL TQ ALCANZADO" )
   END_RUNG
   RUNG wire#powerrail
      Contact( #"CICLO OP FINALIZADO" )
   END_RUNG wire#w3
   RUNG wire#powerrail
      Contact( #"CICLO CANCELADO" )
   END_RUNG wire#w3
   // the same network as SCL:
   #_w1 := (#"CICLO PO ACTIVO" OR #"CICLO OP ACTIVO") AND NOT #"NIVEL TQ ALCANZADO";
   #"CARGA AGUA TQ" := #_w1 AND (#NIVEL < #"NIVEL PARA CARGA DE AGUA");
   IF #_w1 AND (#NIVEL >= #"NIVEL PARA CARGA DE AGUA") THEN #"NIVEL TQ ALCANZADO" := TRUE; END_IF;
   IF #"CICLO PO FINALIZADO" OR #"CICLO OP FINALIZADO" OR #"CICLO CANCELADO" THEN
       #"NIVEL TQ ALCANZADO" := FALSE;
   END_IF;
END_REGION

REGION Network 9: CARGA DE AGUA
   RUNG wire#powerrail
      Contact( #"CARGA AGUA TQ" )
      I_Contact( #"CICLO PAUSADO" )
      wire#w1
      Coil( #"CARGA DE AGUA" )
   END_RUNG
   RUNG wire#powerrail
      Contact( #"MANUAL CARGA DE AGUA" )
   END_RUNG wire#w1
   // the same network as SCL:
   #"CARGA DE AGUA" := (#"CARGA AGUA TQ" AND NOT #"CICLO PAUSADO") OR #"MANUAL CARGA DE AGUA";
END_REGION

REGION Network 10: PRE OPERATIVO POR TEMPERATURA
   RUNG wire#powerrail
      Contact( #"CICLO PO ACTIVO" )
      Contact( #"NIVEL TQ ALCANZADO" )
      Contact( #"PARAMETROS CICLOS"."TIPO DE CORTE" )
      { S7_Templates := "SrcType := Real" } GE_Contact(in1 := #TEMPERATURAS."TEMPERATURA AGUA", in2 := #"PARAMETROS CICLOS"."TEMPERATURA CORTE PO")
      Coil( #"TEMPERATURA PO ALCANZADA" )
   END_RUNG
   // the same network as SCL:
   #"TEMPERATURA PO ALCANZADA" := #"CICLO PO ACTIVO" AND #"NIVEL TQ ALCANZADO" AND #"PARAMETROS CICLOS"."TIPO DE CORTE" AND (#TEMPERATURAS."TEMPERATURA AGUA" >= #"PARAMETROS CICLOS"."TEMPERATURA CORTE PO");
END_REGION

REGION Network 11: PRE OPERATIVO POR TIEMPO
   "CONVERSOR MIN A MS"("TIEMPO EN MIN" := #"PARAMETROS CICLOS"."TIEMPO CORTE PO",
                        "TIEMPO EN MS" => #"TIEMPO CORTE PO");
   #IEC_Timer_0_Instance(IN := #"CICLO PO ACTIVO" AND #"NIVEL TQ ALCANZADO" AND NOT #"PARAMETROS CICLOS"."TIPO DE CORTE" AND NOT #"CICLO PAUSADO",   // TONR
                         R := NOT #"CICLO PO ACTIVO",
                         PT := #"TIEMPO CORTE PO");
   #"TIEMPO PO ALCANZADO" := #IEC_Timer_0_Instance.Q;
END_REGION

REGION Network 12: CICLO PO FINALIZADO
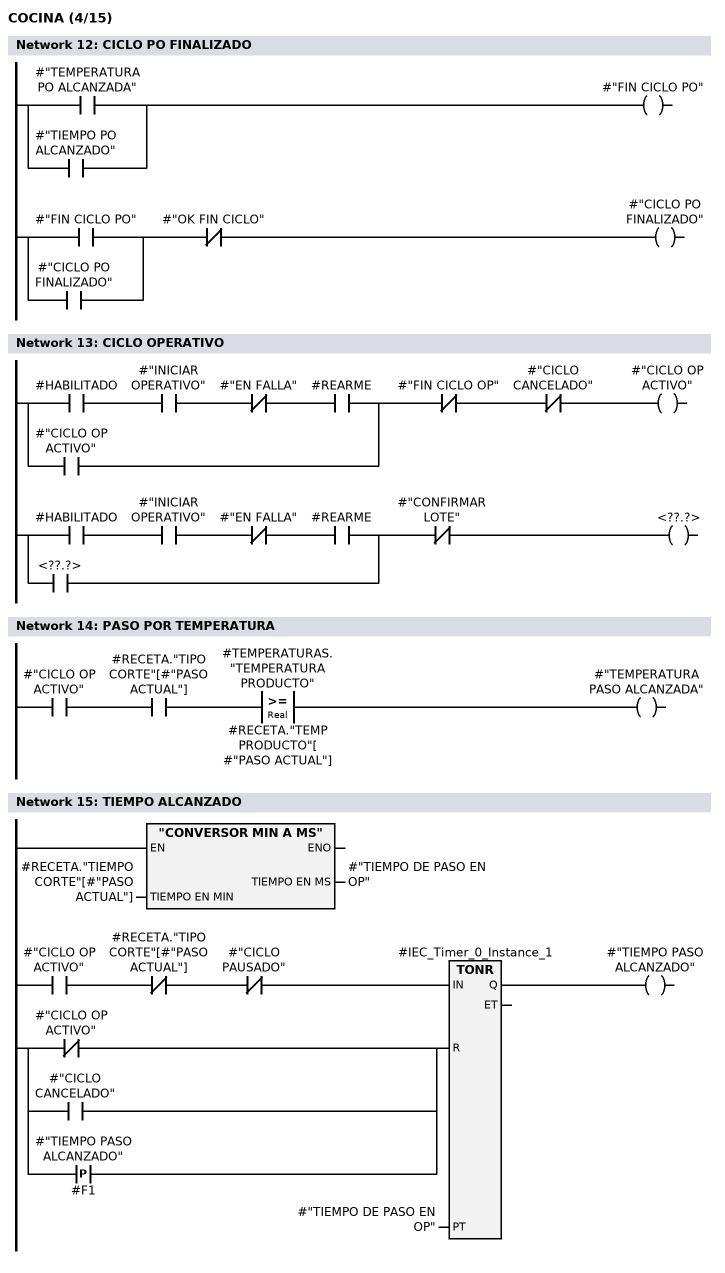
   RUNG wire#powerrail
      Contact( #"TEMPERATURA PO ALCANZADA" )
      wire#w1
      Coil( #"FIN CICLO PO" )
   END_RUNG
   RUNG wire#powerrail
      Contact( #"TIEMPO PO ALCANZADO" )
   END_RUNG wire#w1
   RUNG wire#powerrail
      Contact( #"FIN CICLO PO" )
      wire#w2
      I_Contact( #"OK FIN CICLO" )
      Coil( #"CICLO PO FINALIZADO" )
   END_RUNG
   RUNG wire#powerrail
      Contact( #"CICLO PO FINALIZADO" )
   END_RUNG wire#w2
   // the same network as SCL:
   #"FIN CICLO PO" := #"TEMPERATURA PO ALCANZADA" OR #"TIEMPO PO ALCANZADO";
   #"CICLO PO FINALIZADO" := (#"FIN CICLO PO" OR #"CICLO PO FINALIZADO") AND NOT #"OK FIN CICLO";
END_REGION

REGION Network 13: CICLO OPERATIVO
   RUNG wire#powerrail
      Contact( #HABILITADO )
      Contact( #"INICIAR OPERATIVO" )
      I_Contact( #"EN FALLA" )
      Contact( #REARME )
      wire#w1
      I_Contact( #"FIN CICLO OP" )
      I_Contact( #"CICLO CANCELADO" )
      Coil( #"CICLO OP ACTIVO" )
   END_RUNG
   RUNG wire#powerrail
      Contact( #"CICLO OP ACTIVO" )
   END_RUNG wire#w1
   RUNG wire#powerrail
      Contact( #HABILITADO )
      Contact( #"INICIAR OPERATIVO" )
      I_Contact( #"EN FALLA" )
      Contact( #REARME )
      wire#w2
      I_Contact( #"CONFIRMAR LOTE" )
      Coil(  )
   END_RUNG
   RUNG wire#powerrail
      Contact(  )
   END_RUNG wire#w2
   // the same network as SCL:
   #"CICLO OP ACTIVO" := ((#HABILITADO AND #"INICIAR OPERATIVO" AND NOT #"EN FALLA" AND #REARME) OR #"CICLO OP ACTIVO") AND NOT #"FIN CICLO OP" AND NOT #"CICLO CANCELADO";
   <??.?> := ((#HABILITADO AND #"INICIAR OPERATIVO" AND NOT #"EN FALLA" AND #REARME) OR <??.?>) AND NOT #"CONFIRMAR LOTE";
END_REGION

REGION Network 14: PASO POR TEMPERATURA
   RUNG wire#powerrail
      Contact( #"CICLO OP ACTIVO" )
      Contact( #RECETA."TIPO CORTE"[#"PASO ACTUAL"] )
      { S7_Templates := "SrcType := Real" } GE_Contact(in1 := #TEMPERATURAS."TEMPERATURA PRODUCTO", in2 := #RECETA."TEMP PRODUCTO"[#"PASO ACTUAL"])
      Coil( #"TEMPERATURA PASO ALCANZADA" )
   END_RUNG
   // the same network as SCL:
   #"TEMPERATURA PASO ALCANZADA" := #"CICLO OP ACTIVO" AND #RECETA."TIPO CORTE"[#"PASO ACTUAL"] AND (#TEMPERATURAS."TEMPERATURA PRODUCTO" >= #RECETA."TEMP PRODUCTO"[#"PASO ACTUAL"]);
END_REGION

REGION Network 15: TIEMPO ALCANZADO
   "CONVERSOR MIN A MS"("TIEMPO EN MIN" := #RECETA."TIEMPO CORTE"[#"PASO ACTUAL"],
                        "TIEMPO EN MS" => #"TIEMPO DE PASO EN OP");
   #_w1 := #"TIEMPO PASO ALCANZADO" AND NOT #F1;   // rising edge of #"TIEMPO PASO ALCANZADO"
   #F1 := #"TIEMPO PASO ALCANZADO";
   #IEC_Timer_0_Instance_1(IN := #"CICLO OP ACTIVO" AND NOT #RECETA."TIPO CORTE"[#"PASO ACTUAL"] AND NOT #"CICLO PAUSADO",   // TONR
                           R := NOT #"CICLO OP ACTIVO" OR #"CICLO CANCELADO" OR #_w1,
                           PT := #"TIEMPO DE PASO EN OP");
   #"TIEMPO PASO ALCANZADO" := #IEC_Timer_0_Instance_1.Q;
END_REGION

REGION Network 16: CONTADOR DE PASOS
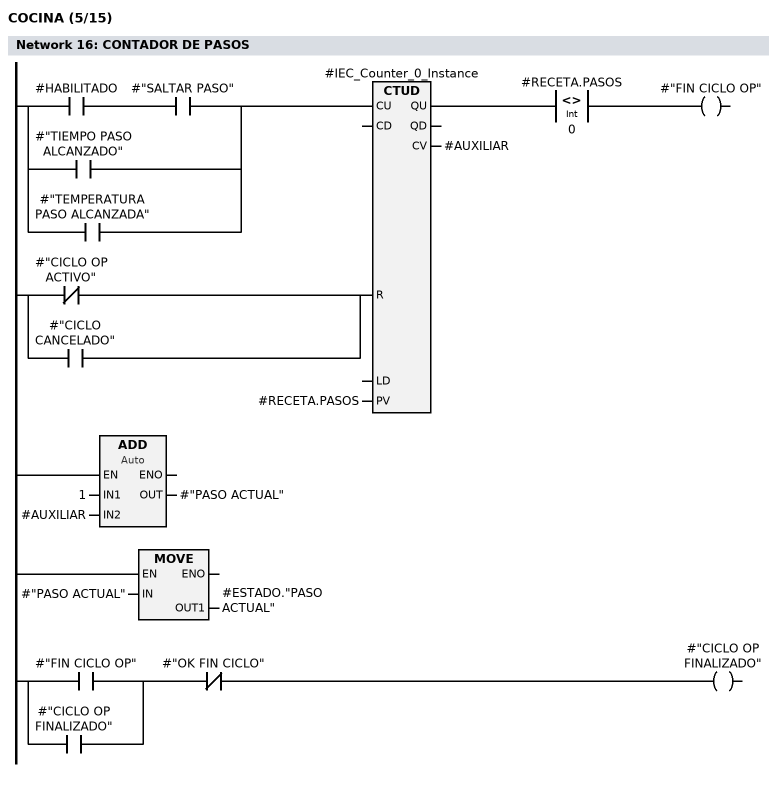
   #IEC_Counter_0_Instance(CU := (#HABILITADO AND #"SALTAR PASO") OR #"TIEMPO PASO ALCANZADO" OR #"TEMPERATURA PASO ALCANZADA",   // CTUD
                           R := NOT #"CICLO OP ACTIVO" OR #"CICLO CANCELADO",
                           PV := #RECETA.PASOS,
                           CV => #AUXILIAR);
   #"FIN CICLO OP" := #IEC_Counter_0_Instance.QU AND (#RECETA.PASOS <> 0);
   #"PASO ACTUAL" := 1 + #AUXILIAR;
   #ESTADO."PASO ACTUAL" := #"PASO ACTUAL";
   #"CICLO OP FINALIZADO" := (#"FIN CICLO OP" OR #"CICLO OP FINALIZADO") AND NOT #"OK FIN CICLO";
END_REGION

REGION Network 17: CONTROL DE TEMPERATURA
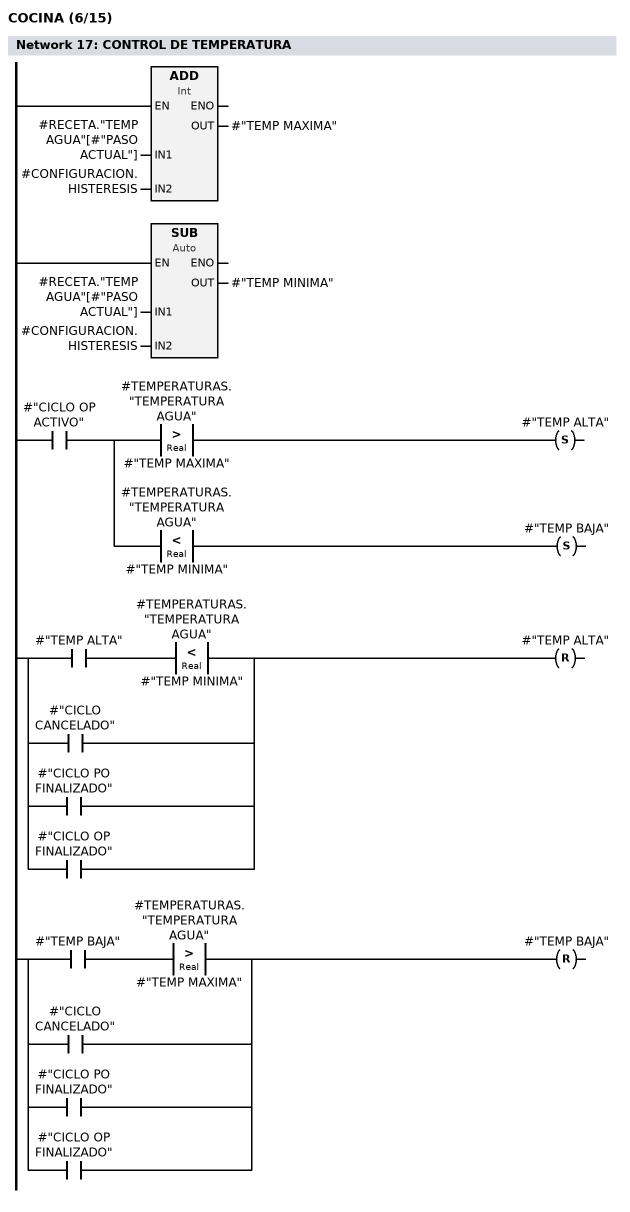
   RUNG wire#powerrail
      { S7_Templates := "SrcType := Int" } Add(in1 := #RECETA."TEMP AGUA"[#"PASO ACTUAL"], in2 := #CONFIGURACION.HISTERESIS, out => #"TEMP MAXIMA")
   END_RUNG
   RUNG wire#powerrail
      Sub(in1 := #RECETA."TEMP AGUA"[#"PASO ACTUAL"], in2 := #CONFIGURACION.HISTERESIS, out => #"TEMP MINIMA")
   END_RUNG
   RUNG wire#powerrail
      Contact( #"CICLO OP ACTIVO" )
      wire#w1
      { S7_Templates := "SrcType := Real" } GT_Contact(in1 := #TEMPERATURAS."TEMPERATURA AGUA", in2 := #"TEMP MAXIMA")
      S_Coil( #"TEMP ALTA" )
   END_RUNG
   RUNG wire#w1
      { S7_Templates := "SrcType := Real" } LT_Contact(in1 := #TEMPERATURAS."TEMPERATURA AGUA", in2 := #"TEMP MINIMA")
      S_Coil( #"TEMP BAJA" )
   END_RUNG
   RUNG wire#powerrail
      Contact( #"TEMP ALTA" )
      { S7_Templates := "SrcType := Real" } LT_Contact(in1 := #TEMPERATURAS."TEMPERATURA AGUA", in2 := #"TEMP MINIMA")
      wire#w2
      R_Coil( #"TEMP ALTA" )
   END_RUNG
   RUNG wire#powerrail
      Contact( #"CICLO CANCELADO" )
   END_RUNG wire#w2
   RUNG wire#powerrail
      Contact( #"CICLO PO FINALIZADO" )
   END_RUNG wire#w2
   RUNG wire#powerrail
      Contact( #"CICLO OP FINALIZADO" )
   END_RUNG wire#w2
   RUNG wire#powerrail
      Contact( #"TEMP BAJA" )
      { S7_Templates := "SrcType := Real" } GT_Contact(in1 := #TEMPERATURAS."TEMPERATURA AGUA", in2 := #"TEMP MAXIMA")
      wire#w3
      R_Coil( #"TEMP BAJA" )
   END_RUNG
   RUNG wire#powerrail
      Contact( #"CICLO CANCELADO" )
   END_RUNG wire#w3
   RUNG wire#powerrail
      Contact( #"CICLO PO FINALIZADO" )
   END_RUNG wire#w3
   RUNG wire#powerrail
      Contact( #"CICLO OP FINALIZADO" )
   END_RUNG wire#w3
   // the same network as SCL:
   #"TEMP MAXIMA" := #RECETA."TEMP AGUA"[#"PASO ACTUAL"] + #CONFIGURACION.HISTERESIS;
   #"TEMP MINIMA" := #RECETA."TEMP AGUA"[#"PASO ACTUAL"] - #CONFIGURACION.HISTERESIS;
   IF #"CICLO OP ACTIVO" AND (#TEMPERATURAS."TEMPERATURA AGUA" > #"TEMP MAXIMA") THEN
       #"TEMP ALTA" := TRUE;
   END_IF;
   IF #"CICLO OP ACTIVO" AND (#TEMPERATURAS."TEMPERATURA AGUA" < #"TEMP MINIMA") THEN
       #"TEMP BAJA" := TRUE;
   END_IF;
   IF (#"TEMP ALTA" AND (#TEMPERATURAS."TEMPERATURA AGUA" < #"TEMP MINIMA")) OR #"CICLO CANCELADO" OR #"CICLO PO FINALIZADO" OR #"CICLO OP FINALIZADO" THEN
       #"TEMP ALTA" := FALSE;
   END_IF;
   IF (#"TEMP BAJA" AND (#TEMPERATURAS."TEMPERATURA AGUA" > #"TEMP MAXIMA")) OR #"CICLO CANCELADO" OR #"CICLO PO FINALIZADO" OR #"CICLO OP FINALIZADO" THEN
       #"TEMP BAJA" := FALSE;
   END_IF;
END_REGION

REGION Network 18: ACTIVACION ACTUADORES
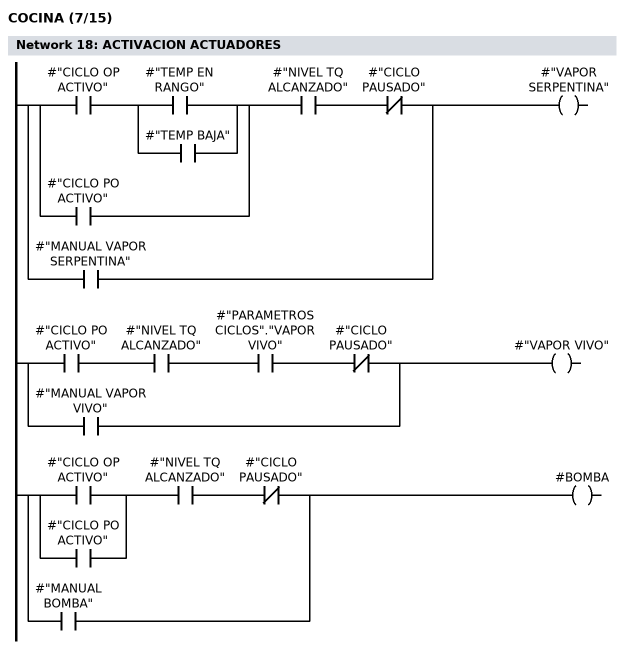
   RUNG wire#powerrail
      Contact( #"CICLO OP ACTIVO" )
      wire#w1
      Contact( #"TEMP EN RANGO" )
      wire#w2
      Contact( #"NIVEL TQ ALCANZADO" )
      I_Contact( #"CICLO PAUSADO" )
      wire#w3
      Coil( #"VAPOR SERPENTINA" )
   END_RUNG
   RUNG wire#w1
      Contact( #"TEMP BAJA" )
   END_RUNG wire#w2
   RUNG wire#powerrail
      Contact( #"CICLO PO ACTIVO" )
   END_RUNG wire#w2
   RUNG wire#powerrail
      Contact( #"MANUAL VAPOR SERPENTINA" )
   END_RUNG wire#w3
   RUNG wire#powerrail
      Contact( #"CICLO PO ACTIVO" )
      Contact( #"NIVEL TQ ALCANZADO" )
      Contact( #"PARAMETROS CICLOS"."VAPOR VIVO" )
      I_Contact( #"CICLO PAUSADO" )
      wire#w4
      Coil( #"VAPOR VIVO" )
   END_RUNG
   RUNG wire#powerrail
      Contact( #"MANUAL VAPOR VIVO" )
   END_RUNG wire#w4
   RUNG wire#powerrail
      Contact( #"CICLO OP ACTIVO" )
      wire#w5
      Contact( #"NIVEL TQ ALCANZADO" )
      I_Contact( #"CICLO PAUSADO" )
      wire#w6
      Coil( #BOMBA )
   END_RUNG
   RUNG wire#powerrail
      Contact( #"CICLO PO ACTIVO" )
   END_RUNG wire#w5
   RUNG wire#powerrail
      Contact( #"MANUAL BOMBA" )
   END_RUNG wire#w6
   // the same network as SCL:
   #"VAPOR SERPENTINA" := (((#"CICLO OP ACTIVO" AND (#"TEMP EN RANGO" OR #"TEMP BAJA")) OR #"CICLO PO ACTIVO") AND #"NIVEL TQ ALCANZADO" AND NOT #"CICLO PAUSADO") OR #"MANUAL VAPOR SERPENTINA";
   #"VAPOR VIVO" := (#"CICLO PO ACTIVO" AND #"NIVEL TQ ALCANZADO" AND #"PARAMETROS CICLOS"."VAPOR VIVO" AND NOT #"CICLO PAUSADO") OR #"MANUAL VAPOR VIVO";
   #BOMBA := ((#"CICLO OP ACTIVO" OR #"CICLO PO ACTIVO") AND #"NIVEL TQ ALCANZADO" AND NOT #"CICLO PAUSADO") OR #"MANUAL BOMBA";
END_REGION

REGION Network 19: VISIBILIDAD HMI
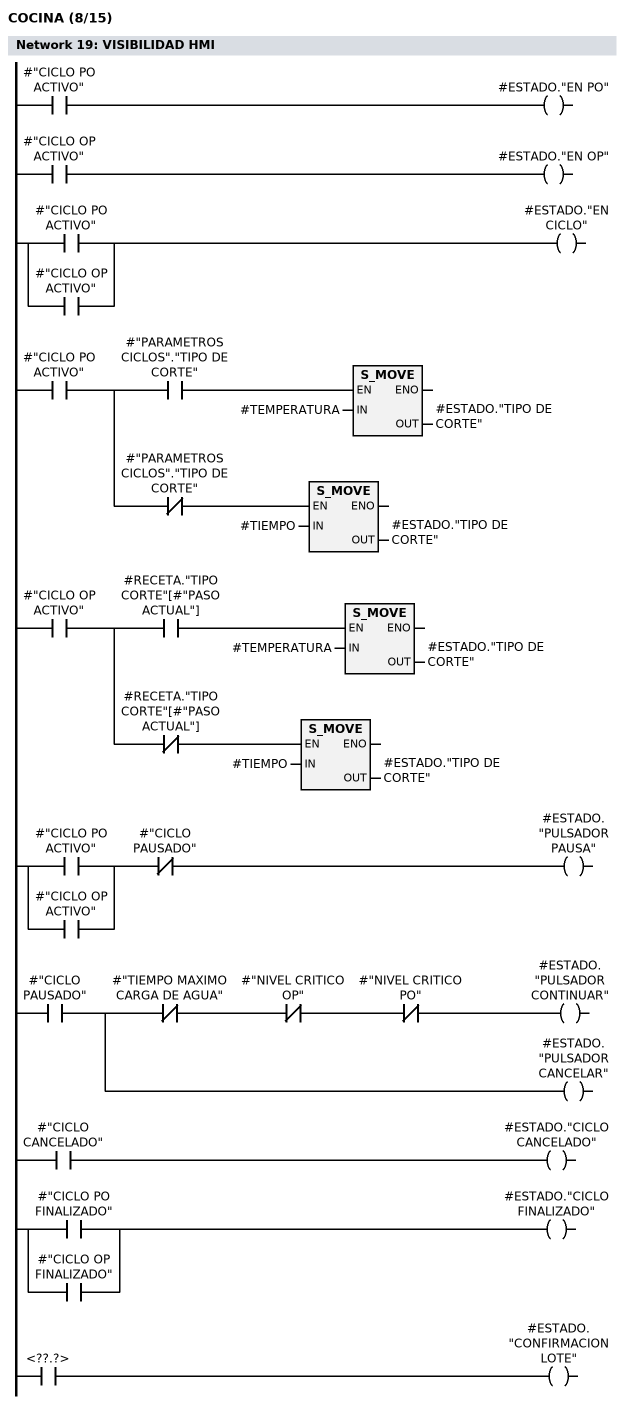
   RUNG wire#powerrail
      Contact( #"CICLO PO ACTIVO" )
      Coil( #ESTADO."EN PO" )
   END_RUNG
   RUNG wire#powerrail
      Contact( #"CICLO OP ACTIVO" )
      Coil( #ESTADO."EN OP" )
   END_RUNG
   RUNG wire#powerrail
      Contact( #"CICLO PO ACTIVO" )
      wire#w1
      Coil( #ESTADO."EN CICLO" )
   END_RUNG
   RUNG wire#powerrail
      Contact( #"CICLO OP ACTIVO" )
   END_RUNG wire#w1
   RUNG wire#powerrail
      Contact( #"CICLO PO ACTIVO" )
      wire#w2
      Contact( #"PARAMETROS CICLOS"."TIPO DE CORTE" )
      S_Move(in := #TEMPERATURA, out => #ESTADO."TIPO DE CORTE")
   END_RUNG
   RUNG wire#w2
      I_Contact( #"PARAMETROS CICLOS"."TIPO DE CORTE" )
      S_Move(in := #TIEMPO, out => #ESTADO."TIPO DE CORTE")
   END_RUNG
   RUNG wire#powerrail
      Contact( #"CICLO OP ACTIVO" )
      wire#w3
      Contact( #RECETA."TIPO CORTE"[#"PASO ACTUAL"] )
      S_Move(in := #TEMPERATURA, out => #ESTADO."TIPO DE CORTE")
   END_RUNG
   RUNG wire#w3
      I_Contact( #RECETA."TIPO CORTE"[#"PASO ACTUAL"] )
      S_Move(in := #TIEMPO, out => #ESTADO."TIPO DE CORTE")
   END_RUNG
   RUNG wire#powerrail
      Contact( #"CICLO PO ACTIVO" )
      wire#w4
      I_Contact( #"CICLO PAUSADO" )
      Coil( #ESTADO."PULSADOR PAUSA" )
   END_RUNG
   RUNG wire#powerrail
      Contact( #"CICLO OP ACTIVO" )
   END_RUNG wire#w4
   RUNG wire#powerrail
      Contact( #"CICLO PAUSADO" )
      wire#w5
      I_Contact( #"TIEMPO MAXIMO CARGA DE AGUA" )
      I_Contact( #"NIVEL CRITICO OP" )
      I_Contact( #"NIVEL CRITICO PO" )
      Coil( #ESTADO."PULSADOR CONTINUAR" )
   END_RUNG
   RUNG wire#w5
      Coil( #ESTADO."PULSADOR CANCELAR" )
   END_RUNG
   RUNG wire#powerrail
      Contact( #"CICLO CANCELADO" )
      Coil( #ESTADO."CICLO CANCELADO" )
   END_RUNG
   RUNG wire#powerrail
      Contact( #"CICLO PO FINALIZADO" )
      wire#w6
      Coil( #ESTADO."CICLO FINALIZADO" )
   END_RUNG
   RUNG wire#powerrail
      Contact( #"CICLO OP FINALIZADO" )
   END_RUNG wire#w6
   RUNG wire#powerrail
      Contact(  )
      Coil( #ESTADO."CONFIRMACION LOTE" )
   END_RUNG
   // the same network as SCL:
   // no checked SCL form for this network; see the picture
END_REGION

REGION Network 20: ESTADO EQUIPO (COLOR HMI EN PRINCIPAL)
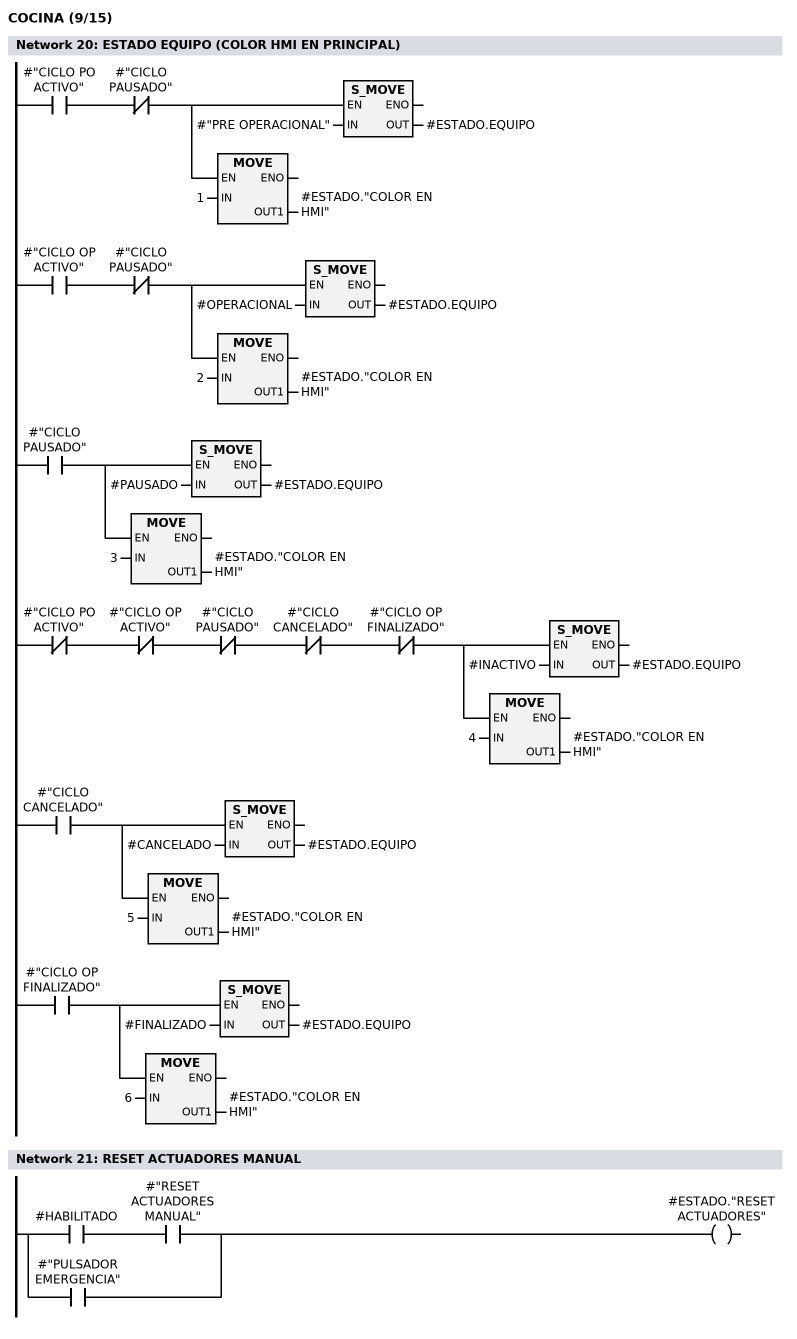
   RUNG wire#powerrail
      Contact( #"CICLO PO ACTIVO" )
      I_Contact( #"CICLO PAUSADO" )
      wire#w1
      S_Move(in := #"PRE OPERACIONAL", out => #ESTADO.EQUIPO)
   END_RUNG
   RUNG wire#w1
      Move(in := 1, out1 => #ESTADO."COLOR EN HMI")
   END_RUNG
   RUNG wire#powerrail
      Contact( #"CICLO OP ACTIVO" )
      I_Contact( #"CICLO PAUSADO" )
      wire#w2
      S_Move(in := #OPERACIONAL, out => #ESTADO.EQUIPO)
   END_RUNG
   RUNG wire#w2
      Move(in := 2, out1 => #ESTADO."COLOR EN HMI")
   END_RUNG
   RUNG wire#powerrail
      Contact( #"CICLO PAUSADO" )
      wire#w3
      S_Move(in := #PAUSADO, out => #ESTADO.EQUIPO)
   END_RUNG
   RUNG wire#w3
      Move(in := 3, out1 => #ESTADO."COLOR EN HMI")
   END_RUNG
   RUNG wire#powerrail
      I_Contact( #"CICLO PO ACTIVO" )
      I_Contact( #"CICLO OP ACTIVO" )
      I_Contact( #"CICLO PAUSADO" )
      I_Contact( #"CICLO CANCELADO" )
      I_Contact( #"CICLO OP FINALIZADO" )
      wire#w4
      S_Move(in := #INACTIVO, out => #ESTADO.EQUIPO)
   END_RUNG
   RUNG wire#w4
      Move(in := 4, out1 => #ESTADO."COLOR EN HMI")
   END_RUNG
   RUNG wire#powerrail
      Contact( #"CICLO CANCELADO" )
      wire#w5
      S_Move(in := #CANCELADO, out => #ESTADO.EQUIPO)
   END_RUNG
   RUNG wire#w5
      Move(in := 5, out1 => #ESTADO."COLOR EN HMI")
   END_RUNG
   RUNG wire#powerrail
      Contact( #"CICLO OP FINALIZADO" )
      wire#w6
      S_Move(in := #FINALIZADO, out => #ESTADO.EQUIPO)
   END_RUNG
   RUNG wire#w6
      Move(in := 6, out1 => #ESTADO."COLOR EN HMI")
   END_RUNG
   // the same network as SCL:
   IF #"CICLO PO ACTIVO" AND NOT #"CICLO PAUSADO" THEN
       #ESTADO.EQUIPO := #"PRE OPERACIONAL";
       #ESTADO."COLOR EN HMI" := 1;
   END_IF;
   IF #"CICLO OP ACTIVO" AND NOT #"CICLO PAUSADO" THEN
       #ESTADO.EQUIPO := #OPERACIONAL;
       #ESTADO."COLOR EN HMI" := 2;
   END_IF;
   IF #"CICLO PAUSADO" THEN
       #ESTADO.EQUIPO := #PAUSADO;
       #ESTADO."COLOR EN HMI" := 3;
   END_IF;
   IF NOT #"CICLO PO ACTIVO" AND NOT #"CICLO OP ACTIVO" AND NOT #"CICLO PAUSADO" AND NOT #"CICLO CANCELADO" AND NOT #"CICLO OP FINALIZADO" THEN
       #ESTADO.EQUIPO := #INACTIVO;
       #ESTADO."COLOR EN HMI" := 4;
   END_IF;
   IF #"CICLO CANCELADO" THEN
       #ESTADO.EQUIPO := #CANCELADO;
       #ESTADO."COLOR EN HMI" := 5;
   END_IF;
   IF #"CICLO OP FINALIZADO" THEN
       #ESTADO.EQUIPO := #FINALIZADO;
       #ESTADO."COLOR EN HMI" := 6;
   END_IF;
END_REGION

REGION Network 21: RESET ACTUADORES MANUAL
   RUNG wire#powerrail
      Contact( #HABILITADO )
      Contact( #"RESET ACTUADORES MANUAL" )
      wire#w1
      Coil( #ESTADO."RESET ACTUADORES" )
   END_RUNG
   RUNG wire#powerrail
      Contact( #"PULSADOR EMERGENCIA" )
   END_RUNG wire#w1
   // the same network as SCL:
   #ESTADO."RESET ACTUADORES" := (#HABILITADO AND #"RESET ACTUADORES MANUAL") OR #"PULSADOR EMERGENCIA";
END_REGION

REGION Network 22: ACTUADORES MANUALES ACTIVOS
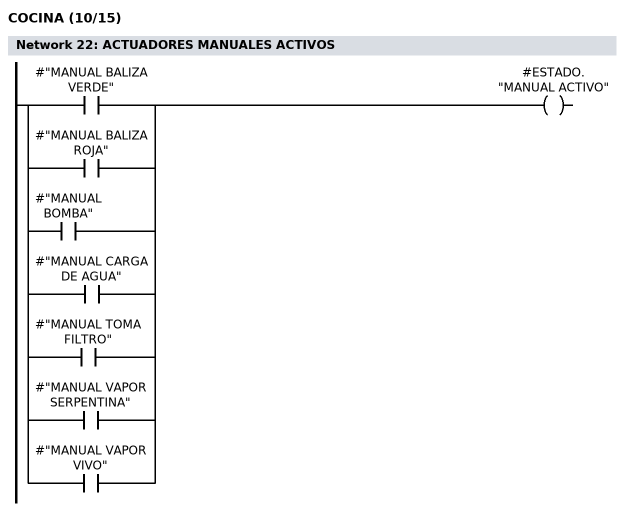
   RUNG wire#powerrail
      Contact( #"MANUAL BALIZA VERDE" )
      wire#w1
      Coil( #ESTADO."MANUAL ACTIVO" )
   END_RUNG
   RUNG wire#powerrail
      Contact( #"MANUAL BALIZA ROJA" )
   END_RUNG wire#w1
   RUNG wire#powerrail
      Contact( #"MANUAL BOMBA" )
   END_RUNG wire#w1
   RUNG wire#powerrail
      Contact( #"MANUAL CARGA DE AGUA" )
   END_RUNG wire#w1
   RUNG wire#powerrail
      Contact( #"MANUAL TOMA FILTRO" )
   END_RUNG wire#w1
   RUNG wire#powerrail
      Contact( #"MANUAL VAPOR SERPENTINA" )
   END_RUNG wire#w1
   RUNG wire#powerrail
      Contact( #"MANUAL VAPOR VIVO" )
   END_RUNG wire#w1
   // the same network as SCL:
   #ESTADO."MANUAL ACTIVO" := #"MANUAL BALIZA VERDE" OR #"MANUAL BALIZA ROJA" OR #"MANUAL BOMBA" OR #"MANUAL CARGA DE AGUA" OR #"MANUAL TOMA FILTRO" OR #"MANUAL VAPOR SERPENTINA" OR #"MANUAL VAPOR VIVO";
END_REGION

REGION Network 23: SALIDAS ACTIVAS PARA VISUALIZAR EN HMI
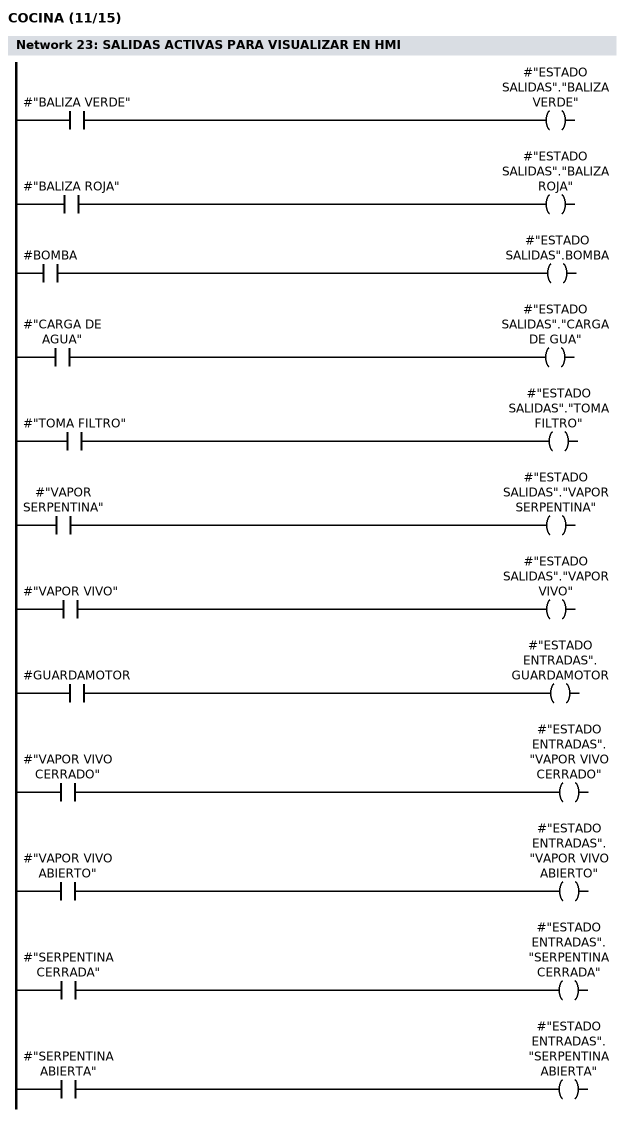
   RUNG wire#powerrail
      Contact( #"BALIZA VERDE" )
      Coil( #"ESTADO SALIDAS"."BALIZA VERDE" )
   END_RUNG
   RUNG wire#powerrail
      Contact( #"BALIZA ROJA" )
      Coil( #"ESTADO SALIDAS"."BALIZA ROJA" )
   END_RUNG
   RUNG wire#powerrail
      Contact( #BOMBA )
      Coil( #"ESTADO SALIDAS".BOMBA )
   END_RUNG
   RUNG wire#powerrail
      Contact( #"CARGA DE AGUA" )
      Coil( #"ESTADO SALIDAS"."CARGA DE GUA" )
   END_RUNG
   RUNG wire#powerrail
      Contact( #"TOMA FILTRO" )
      Coil( #"ESTADO SALIDAS"."TOMA FILTRO" )
   END_RUNG
   RUNG wire#powerrail
      Contact( #"VAPOR SERPENTINA" )
      Coil( #"ESTADO SALIDAS"."VAPOR SERPENTINA" )
   END_RUNG
   RUNG wire#powerrail
      Contact( #"VAPOR VIVO" )
      Coil( #"ESTADO SALIDAS"."VAPOR VIVO" )
   END_RUNG
   RUNG wire#powerrail
      Contact( #GUARDAMOTOR )
      Coil( #"ESTADO ENTRADAS".GUARDAMOTOR )
   END_RUNG
   RUNG wire#powerrail
      Contact( #"VAPOR VIVO CERRADO" )
      Coil( #"ESTADO ENTRADAS"."VAPOR VIVO CERRADO" )
   END_RUNG
   RUNG wire#powerrail
      Contact( #"VAPOR VIVO ABIERTO" )
      Coil( #"ESTADO ENTRADAS"."VAPOR VIVO ABIERTO" )
   END_RUNG
   RUNG wire#powerrail
      Contact( #"SERPENTINA CERRADA" )
      Coil( #"ESTADO ENTRADAS"."SERPENTINA CERRADA" )
   END_RUNG
   RUNG wire#powerrail
      Contact( #"SERPENTINA ABIERTA" )
      Coil( #"ESTADO ENTRADAS"."SERPENTINA ABIERTA" )
   END_RUNG
   // the same network as SCL:
   #"ESTADO SALIDAS"."BALIZA VERDE" := #"BALIZA VERDE";
   #"ESTADO SALIDAS"."BALIZA ROJA" := #"BALIZA ROJA";
   #"ESTADO SALIDAS".BOMBA := #BOMBA;
   #"ESTADO SALIDAS"."CARGA DE GUA" := #"CARGA DE AGUA";
   #"ESTADO SALIDAS"."TOMA FILTRO" := #"TOMA FILTRO";
   #"ESTADO SALIDAS"."VAPOR SERPENTINA" := #"VAPOR SERPENTINA";
   #"ESTADO SALIDAS"."VAPOR VIVO" := #"VAPOR VIVO";
   #"ESTADO ENTRADAS".GUARDAMOTOR := #GUARDAMOTOR;
   #"ESTADO ENTRADAS"."VAPOR VIVO CERRADO" := #"VAPOR VIVO CERRADO";
   #"ESTADO ENTRADAS"."VAPOR VIVO ABIERTO" := #"VAPOR VIVO ABIERTO";
   #"ESTADO ENTRADAS"."SERPENTINA CERRADA" := #"SERPENTINA CERRADA";
   #"ESTADO ENTRADAS"."SERPENTINA ABIERTA" := #"SERPENTINA ABIERTA";
END_REGION

REGION Network 24: SEÑALIZACIONES
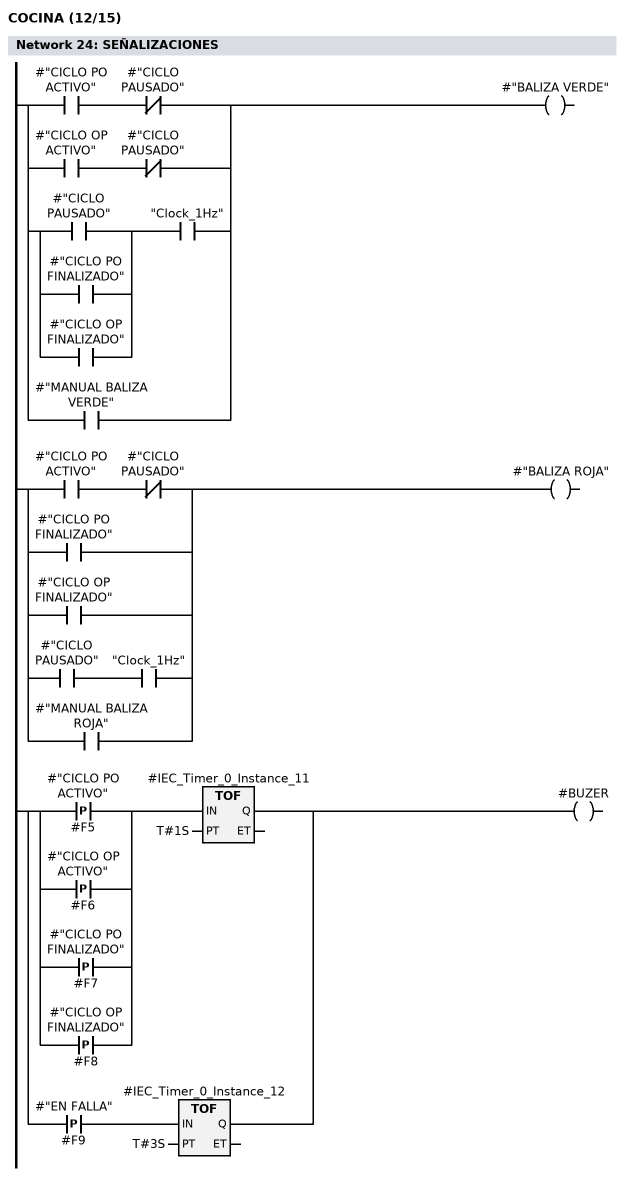
   #"BALIZA VERDE" := (#"CICLO PO ACTIVO" AND NOT #"CICLO PAUSADO") OR (#"CICLO OP ACTIVO" AND NOT #"CICLO PAUSADO") OR ((#"CICLO PAUSADO" OR #"CICLO PO FINALIZADO" OR #"CICLO OP FINALIZADO") AND "Clock_1Hz") OR #"MANUAL BALIZA VERDE";
   #"BALIZA ROJA" := (#"CICLO PO ACTIVO" AND NOT #"CICLO PAUSADO") OR #"CICLO PO FINALIZADO" OR #"CICLO OP FINALIZADO" OR (#"CICLO PAUSADO" AND "Clock_1Hz") OR #"MANUAL BALIZA ROJA";
   #_w1 := #"CICLO PO ACTIVO" AND NOT #F5;   // rising edge of #"CICLO PO ACTIVO"
   #F5 := #"CICLO PO ACTIVO";
   #_w2 := #"CICLO OP ACTIVO" AND NOT #F6;   // rising edge of #"CICLO OP ACTIVO"
   #F6 := #"CICLO OP ACTIVO";
   #_w3 := #"CICLO PO FINALIZADO" AND NOT #F7;   // rising edge of #"CICLO PO FINALIZADO"
   #F7 := #"CICLO PO FINALIZADO";
   #_w4 := #"CICLO OP FINALIZADO" AND NOT #F8;   // rising edge of #"CICLO OP FINALIZADO"
   #F8 := #"CICLO OP FINALIZADO";
   #IEC_Timer_0_Instance_11(IN := #_w1 OR #_w2 OR #_w3 OR #_w4, PT := T#1S);   // TOF
   #_w5 := #"EN FALLA" AND NOT #F9;   // rising edge of #"EN FALLA"
   #F9 := #"EN FALLA";
   #IEC_Timer_0_Instance_12(IN := #_w5, PT := T#3S);   // TOF
   #BUZER := #IEC_Timer_0_Instance_11.Q OR #IEC_Timer_0_Instance_12.Q;
END_REGION

REGION Network 25: TEMPERATURA FUERA DE RANGO
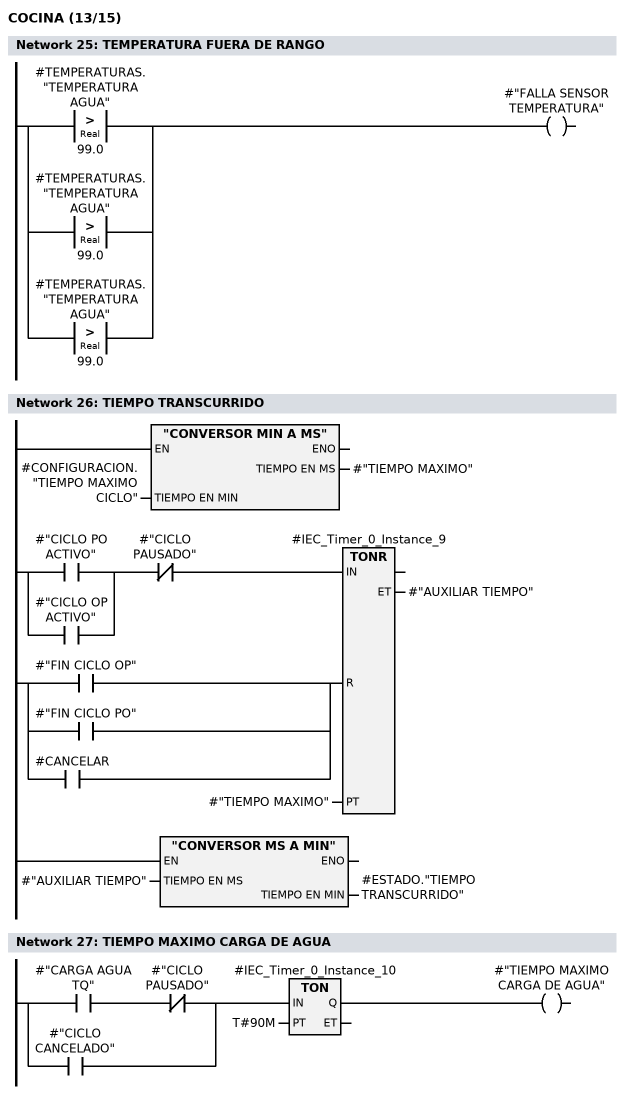
   RUNG wire#powerrail
      { S7_Templates := "SrcType := Real" } GT_Contact(in1 := #TEMPERATURAS."TEMPERATURA AGUA", in2 := 99.0)
      wire#w1
      Coil( #"FALLA SENSOR TEMPERATURA" )
   END_RUNG
   RUNG wire#powerrail
      { S7_Templates := "SrcType := Real" } GT_Contact(in1 := #TEMPERATURAS."TEMPERATURA AGUA", in2 := 99.0)
   END_RUNG wire#w1
   RUNG wire#powerrail
      { S7_Templates := "SrcType := Real" } GT_Contact(in1 := #TEMPERATURAS."TEMPERATURA AGUA", in2 := 99.0)
   END_RUNG wire#w1
   // the same network as SCL:
   #"FALLA SENSOR TEMPERATURA" := (#TEMPERATURAS."TEMPERATURA AGUA" > 99.0) OR (#TEMPERATURAS."TEMPERATURA AGUA" > 99.0) OR (#TEMPERATURAS."TEMPERATURA AGUA" > 99.0);
END_REGION

REGION Network 26: TIEMPO TRANSCURRIDO
   "CONVERSOR MIN A MS"("TIEMPO EN MIN" := #CONFIGURACION."TIEMPO MAXIMO CICLO",
                        "TIEMPO EN MS" => #"TIEMPO MAXIMO");
   #IEC_Timer_0_Instance_9(IN := (#"CICLO PO ACTIVO" OR #"CICLO OP ACTIVO") AND NOT #"CICLO PAUSADO",   // TONR
                           R := #"FIN CICLO OP" OR #"FIN CICLO PO" OR #CANCELAR,
                           PT := #"TIEMPO MAXIMO",
                           ET => #"AUXILIAR TIEMPO");
   "CONVERSOR MS A MIN"("TIEMPO EN MS" := #"AUXILIAR TIEMPO", "TIEMPO EN MIN" => #ESTADO."TIEMPO TRANSCURRIDO");
END_REGION

REGION Network 27: TIEMPO MAXIMO CARGA DE AGUA
   #IEC_Timer_0_Instance_10(IN := (#"CARGA AGUA TQ" AND NOT #"CICLO PAUSADO") OR #"CICLO CANCELADO",   // TON
                           PT := T#90M);
   #"TIEMPO MAXIMO CARGA DE AGUA" := #IEC_Timer_0_Instance_10.Q;
END_REGION

REGION Network 28: NIVELES CRITICOS
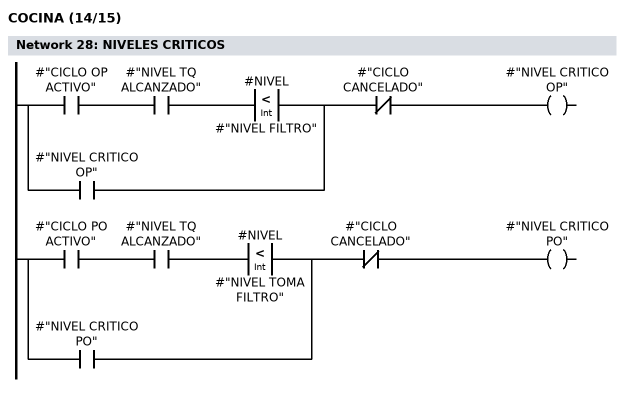
   RUNG wire#powerrail
      Contact( #"CICLO OP ACTIVO" )
      Contact( #"NIVEL TQ ALCANZADO" )
      { S7_Templates := "SrcType := Int" } LT_Contact(in1 := #NIVEL, in2 := #"NIVEL FILTRO")
      wire#w1
      I_Contact( #"CICLO CANCELADO" )
      Coil( #"NIVEL CRITICO OP" )
   END_RUNG
   RUNG wire#powerrail
      Contact( #"NIVEL CRITICO OP" )
   END_RUNG wire#w1
   RUNG wire#powerrail
      Contact( #"CICLO PO ACTIVO" )
      Contact( #"NIVEL TQ ALCANZADO" )
      { S7_Templates := "SrcType := Int" } LT_Contact(in1 := #NIVEL, in2 := #"NIVEL TOMA FILTRO")
      wire#w2
      I_Contact( #"CICLO CANCELADO" )
      Coil( #"NIVEL CRITICO PO" )
   END_RUNG
   RUNG wire#powerrail
      Contact( #"NIVEL CRITICO PO" )
   END_RUNG wire#w2
   // the same network as SCL:
   #"NIVEL CRITICO OP" := ((#"CICLO OP ACTIVO" AND #"NIVEL TQ ALCANZADO" AND (#NIVEL < #"NIVEL FILTRO")) OR #"NIVEL CRITICO OP") AND NOT #"CICLO CANCELADO";
   #"NIVEL CRITICO PO" := ((#"CICLO PO ACTIVO" AND #"NIVEL TQ ALCANZADO" AND (#NIVEL < #"NIVEL TOMA FILTRO")) OR #"NIVEL CRITICO PO") AND NOT #"CICLO CANCELADO";
END_REGION

REGION Network 29: ALARMAS
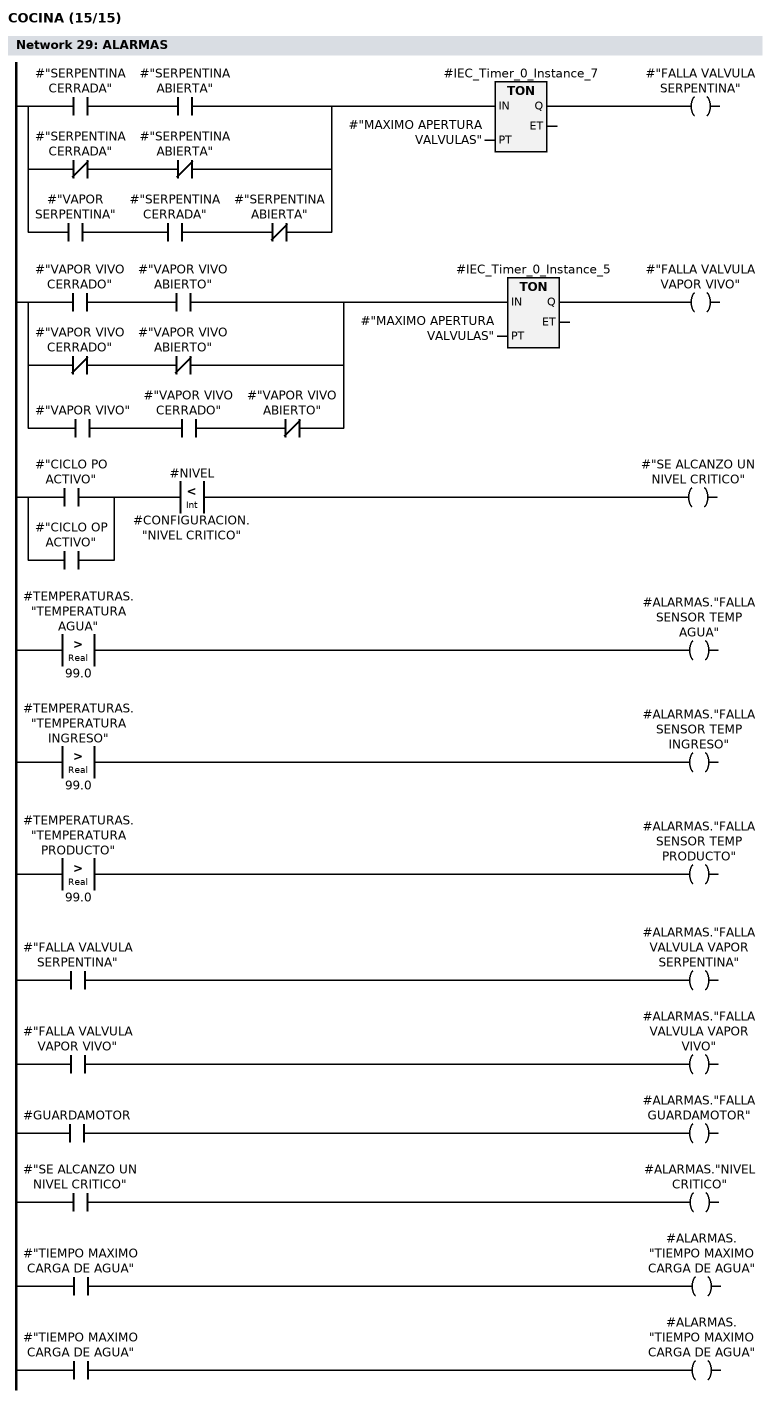
   #IEC_Timer_0_Instance_7(IN := (#"SERPENTINA CERRADA" AND #"SERPENTINA ABIERTA") OR (NOT #"SERPENTINA CERRADA" AND NOT #"SERPENTINA ABIERTA") OR (#"VAPOR SERPENTINA" AND #"SERPENTINA CERRADA" AND NOT #"SERPENTINA ABIERTA"),   // TON
                           PT := #"MAXIMO APERTURA VALVULAS");
   #"FALLA VALVULA SERPENTINA" := #IEC_Timer_0_Instance_7.Q;
   #IEC_Timer_0_Instance_5(IN := (#"VAPOR VIVO CERRADO" AND #"VAPOR VIVO ABIERTO") OR (NOT #"VAPOR VIVO CERRADO" AND NOT #"VAPOR VIVO ABIERTO") OR (#"VAPOR VIVO" AND #"VAPOR VIVO CERRADO" AND NOT #"VAPOR VIVO ABIERTO"),   // TON
                           PT := #"MAXIMO APERTURA VALVULAS");
   #"FALLA VALVULA VAPOR VIVO" := #IEC_Timer_0_Instance_5.Q;
   #"SE ALCANZO UN NIVEL CRITICO" := (#"CICLO PO ACTIVO" OR #"CICLO OP ACTIVO") AND (#NIVEL < #CONFIGURACION."NIVEL CRITICO");
   #ALARMAS."FALLA SENSOR TEMP AGUA" := #TEMPERATURAS."TEMPERATURA AGUA" > 99.0;
   #ALARMAS."FALLA SENSOR TEMP INGRESO" := #TEMPERATURAS."TEMPERATURA INGRESO" > 99.0;
   #ALARMAS."FALLA SENSOR TEMP PRODUCTO" := #TEMPERATURAS."TEMPERATURA PRODUCTO" > 99.0;
   #ALARMAS."FALLA VALVULA VAPOR SERPENTINA" := #"FALLA VALVULA SERPENTINA";
   #ALARMAS."FALLA VALVULA VAPOR VIVO" := #"FALLA VALVULA VAPOR VIVO";
   #ALARMAS."FALLA GUARDAMOTOR" := #GUARDAMOTOR;
   #ALARMAS."NIVEL CRITICO" := #"SE ALCANZO UN NIVEL CRITICO";
   #ALARMAS."TIEMPO MAXIMO CARGA DE AGUA" := #"TIEMPO MAXIMO CARGA DE AGUA";
   #ALARMAS."TIEMPO MAXIMO CARGA DE AGUA" := #"TIEMPO MAXIMO CARGA DE AGUA";
END_REGION
END_FUNCTION_BLOCK

FUNCTION_BLOCK "SEGURIDAD BLOQUEO EQUIPOS"   // FB6, LAD
{ S7_Optimized_Access := 'TRUE' }
VERSION : 0.1
   VAR_INPUT
      "OK CODIGO INGRESADO" : Bool;
      "CONTRASEÑA INGRESADA" : Int;
   END_VAR
   VAR_OUTPUT
      "BLOQUEAR EQUIPOS" : Bool;
      "DIAS TRANSCURRIDOS" : Int;
      "IMAGEN BLOQUEO" : Int;
      "DIAS RESTANTES" : Int;
      "HABILITACION ADVERTENCIA" : Bool;
      "CONTRASEÑA ANTERIOR" : DInt := 1040;
      "CONTRASEÑA ACTUAL" : Int;
      "CONTRASEÑA CORRECTA" : Bool;
      "CONTRASEÑA INCORRECTA" : Bool;
   END_VAR
   VAR
      IEC_Timer_0_Instance : TONR_TIME;
   END_VAR
   VAR RETAIN
      IEC_Counter_0_Instance : CTU_INT;
      "TIEMPO CUMPLIDO PARA BLOQUEO" : Bool;
   END_VAR
   VAR
      RESET : Bool;
      F1 : Bool;
      F2 : Bool;
      CONTR : DInt;
      IEC_Timer_0_Instance_1 : TOF_TIME;
      IEC_Timer_0_Instance_2 : TOF_TIME;
   END_VAR
   VAR_TEMP   // added for the SCL form of the ladder/FBD networks
      _w1 : Bool;
   END_VAR
BEGIN

REGION Network 1
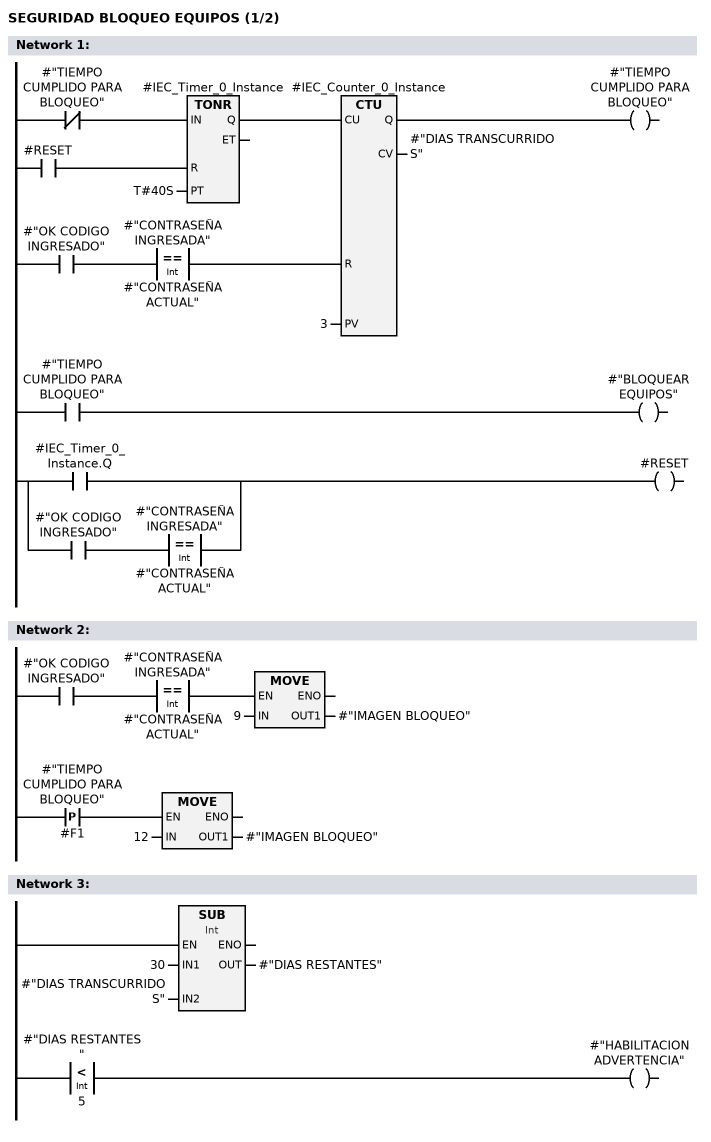
   #IEC_Timer_0_Instance(IN := NOT #"TIEMPO CUMPLIDO PARA BLOQUEO", R := #RESET, PT := T#40S);   // TONR
   #IEC_Counter_0_Instance(CU := #IEC_Timer_0_Instance.Q,   // CTU
                           R := #"OK CODIGO INGRESADO" AND (#"CONTRASEÑA INGRESADA" = #"CONTRASEÑA ACTUAL"),
                           PV := 3,
                           CV => #"DIAS TRANSCURRIDOS");
   #"TIEMPO CUMPLIDO PARA BLOQUEO" := #IEC_Counter_0_Instance.Q;
   #"BLOQUEAR EQUIPOS" := #"TIEMPO CUMPLIDO PARA BLOQUEO";
   #RESET := #IEC_Timer_0_Instance.Q OR (#"OK CODIGO INGRESADO" AND (#"CONTRASEÑA INGRESADA" = #"CONTRASEÑA ACTUAL"));
END_REGION

REGION Network 2
   RUNG wire#powerrail
      Contact( #"OK CODIGO INGRESADO" )
      { S7_Templates := "SrcType := Int" } EQ_Contact(in1 := #"CONTRASEÑA INGRESADA", in2 := #"CONTRASEÑA ACTUAL")
      Move(in := 9, out1 => #"IMAGEN BLOQUEO")
   END_RUNG
   RUNG wire#powerrail
      P_Contact(operand := #"TIEMPO CUMPLIDO PARA BLOQUEO", bit := #F1)
      Move(in := 12, out1 => #"IMAGEN BLOQUEO")
   END_RUNG
   // the same network as SCL:
   IF #"OK CODIGO INGRESADO" AND (#"CONTRASEÑA INGRESADA" = #"CONTRASEÑA ACTUAL") THEN
       #"IMAGEN BLOQUEO" := 9;
   END_IF;
   #_w1 := #"TIEMPO CUMPLIDO PARA BLOQUEO" AND NOT #F1;   // rising edge of #"TIEMPO CUMPLIDO PARA BLOQUEO"
   #F1 := #"TIEMPO CUMPLIDO PARA BLOQUEO";
   IF #_w1 THEN #"IMAGEN BLOQUEO" := 12; END_IF;
END_REGION

REGION Network 3
   RUNG wire#powerrail
      { S7_Templates := "SrcType := Int" } Sub(in1 := 30, in2 := #"DIAS TRANSCURRIDOS", out => #"DIAS RESTANTES")
   END_RUNG
   RUNG wire#powerrail
      { S7_Templates := "SrcType := Int" } LT_Contact(in1 := #"DIAS RESTANTES", in2 := 5)
      Coil( #"HABILITACION ADVERTENCIA" )
   END_RUNG
   // the same network as SCL:
   #"DIAS RESTANTES" := 30 - #"DIAS TRANSCURRIDOS";
   #"HABILITACION ADVERTENCIA" := #"DIAS RESTANTES" < 5;
END_REGION

REGION Network 4
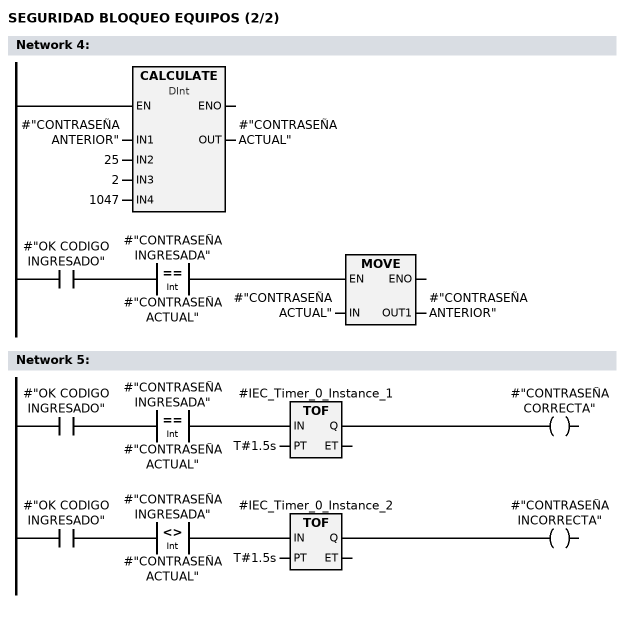
   RUNG wire#powerrail
      { S7_Templates := "SrcType := DInt"; S7_Expression := "((IN1 + IN2)-IN3)+IN4" } Calculate(in1 := #"CONTRASEÑA ANTERIOR", in2 := 25, in3 := 2, in4 := 1047, out => #"CONTRASEÑA ACTUAL")
   END_RUNG
   RUNG wire#powerrail
      Contact( #"OK CODIGO INGRESADO" )
      { S7_Templates := "SrcType := Int" } EQ_Contact(in1 := #"CONTRASEÑA INGRESADA", in2 := #"CONTRASEÑA ACTUAL")
      Move(in := #"CONTRASEÑA ACTUAL", out1 => #"CONTRASEÑA ANTERIOR")
   END_RUNG
   // the same network as SCL:
   #"CONTRASEÑA ACTUAL" := ((#"CONTRASEÑA ANTERIOR" + 25)-2)+1047;
   IF #"OK CODIGO INGRESADO" AND (#"CONTRASEÑA INGRESADA" = #"CONTRASEÑA ACTUAL") THEN
       #"CONTRASEÑA ANTERIOR" := #"CONTRASEÑA ACTUAL";
   END_IF;
END_REGION

REGION Network 5
   #IEC_Timer_0_Instance_1(IN := #"OK CODIGO INGRESADO" AND (#"CONTRASEÑA INGRESADA" = #"CONTRASEÑA ACTUAL"),   // TOF
                           PT := T#1.5s);
   #"CONTRASEÑA CORRECTA" := #IEC_Timer_0_Instance_1.Q;
   #IEC_Timer_0_Instance_2(IN := #"OK CODIGO INGRESADO" AND (#"CONTRASEÑA INGRESADA" <> #"CONTRASEÑA ACTUAL"),   // TOF
                           PT := T#1.5s);
   #"CONTRASEÑA INCORRECTA" := #IEC_Timer_0_Instance_2.Q;
END_REGION
END_FUNCTION_BLOCK

FUNCTION_BLOCK "ENVIO DATOS"   // FB7, SCL
{ S7_Optimized_Access := 'TRUE' }
VERSION : 0.1
   VAR_INPUT
      TEMPERATURAS : Struct
         "TEMPERATURA AGUA" : Real;
         "TEMPERATURA INGRESO" : Real;
         "TEMPERATURA PRODUCTO" : Real;
         "TEMPERATURA AGUA SC" : Real;
         "TEMPERATURA INGRESO SC" : Real;
         "TEMPERATURA PRODUCTO SC" : Real;
      END_STRUCT;
      ESTADO : Int;
      "NIVEL AGUA" : Int;
      RECETA : String;
      "NUM RECETA" : Int;
      "NUMERO EQUIPO" : Int;
      "ESTADO SERPENTINA" : Bool;
      "ESTADO VAPOR VIVO" : Bool;
      TORRES : Int;
      PASOS : Int;
      TIEMPO : DInt;
   END_VAR
   VAR_OUTPUT
      "T AGUA" : Real;
      "T INGRESO" : Real;
      "T PRODUCTO" : Real;
      "ESTADO CICLO" : Int;
      NIVEL : Int;
      "NOMBRE RECETA" : String;
      "NUMERO RECETA" : Int;
      EQUIPO : Int;
      SERPENTINA : Bool;
      "VAPOR VIVO" : Bool;
      "NUMERO TORRES" : Int;
      "CANTIDAD DE PASOS" : Int;
      "TIEMPO TRANSCURRIDO" : DInt;
   END_VAR
BEGIN
   #"T AGUA":= #TEMPERATURAS."TEMPERATURA AGUA";

   #"T INGRESO":= #TEMPERATURAS."TEMPERATURA INGRESO";

   #"T PRODUCTO" := #TEMPERATURAS."TEMPERATURA PRODUCTO";

   #"ESTADO CICLO" := #ESTADO;

   #NIVEL := #"NIVEL AGUA";

   #"NOMBRE RECETA" := #RECETA;

   #"NUMERO RECETA" := #"NUM RECETA";

   #EQUIPO := #"NUMERO EQUIPO";

   #SERPENTINA := #"ESTADO SERPENTINA";

   #"VAPOR VIVO" := #"ESTADO VAPOR VIVO";

   #"NUMERO TORRES" := #TORRES;

   #"CANTIDAD DE PASOS" := #PASOS;

   #"TIEMPO TRANSCURRIDO" := #TIEMPO;
END_FUNCTION_BLOCK

FUNCTION "ESCALADO TEMPERATURAS" : Void   // FC1, LAD
{ S7_Optimized_Access := 'TRUE' }
VERSION : 0.1
   VAR_INPUT
      "DATO PT100" : Int;
      CORRECCION : Real;
   END_VAR
   VAR_OUTPUT
      "TEMPERATURA CORREGIDA" : Real;
      "TEMPERATURA SIN CORREGIR" : Real;
   END_VAR
   VAR_TEMP
      AUXILIAR : Real;
      "SIN CORREGIR" : Real;
   END_VAR
BEGIN

REGION Network 1
